Yaskawa INFORM job: SKRZYNIA_5240_0_STOPNI_1OBR.JBI

/JOB
//NAME SKRZYNIA_5240_0_STOPNI_1OBR
///FOLDERNAME 02-SKRZYNIE_JOBS
//POS
///NPOS 629,629,0,49,4,0
///TOOL 0
///POSTYPE PULSE
///PULSE
C00000=1055,-24125,84372,288,19725,204
C00001=1055,-24125,84372,288,19725,204
C00002=0,-15438,65714,0,-68532,0
C00003=25524,-25821,36823,19654,-58495,38520
C00004=25525,-25816,36822,19654,-58489,38517
C00005=24740,-25233,37027,19126,-58082,38651
C00006=23674,-24366,37359,18410,-57511,38837
C00007=23935,-24587,37271,18586,-57653,38791
C00008=22514,-24691,37230,17505,-57481,39152
C00009=26142,-25637,36881,20127,-58504,38350
C00010=24740,-25232,37025,19127,-58082,38646
C00011=24741,-25229,37025,19127,-58082,38646
C00012=24435,-24991,37114,18923,-57922,38699
C00013=23923,-24572,37275,18578,-57647,38788
C00014=24083,-24706,37224,18686,-57733,38759
C00015=22429,-24825,37180,17430,-57534,39178
C00016=25895,-26212,36688,19885,-58747,38460
C00017=25524,-25821,36823,19654,-58495,38520
C00018=23988,-24960,37134,18595,-57837,38812
C00019=22822,-23954,37534,17811,-57199,39017
C00020=22935,-24057,37491,17887,-57262,38997
C00021=20006,-24258,37408,15644,-56932,39751
C00022=24402,-25289,37013,18874,-58060,38740
C00023=22585,-24665,40358,17164,-59622,30036
C00024=23477,-23257,40205,18030,-58646,29630
C00025=22519,-22398,40568,17384,-58125,29795
C00026=22700,-22567,40495,17506,-58225,29764
C00027=19339,-22794,40398,14955,-57865,30607
C00028=24825,-24328,39798,18931,-59350,29401
C00029=32755,-32613,25711,29640,-48730,33694
C00030=25632,-30899,26166,23992,-46203,35378
C00031=24264,-29862,26497,22996,-45413,35639
C00032=24403,-29974,26459,23097,-45496,35612
C00033=20575,-30233,26374,19602,-44891,36810
C00034=26556,-31526,25988,24663,-46720,35206
C00035=30846,-32795,25752,28021,-48338,30427
C00036=24953,-30697,26306,23444,-45946,31743
C00037=23937,-29910,26558,22702,-45353,31936
C00038=24039,-29993,26530,22778,-45414,31916
C00039=20322,-30240,26449,19379,-44834,33080
C00040=25997,-31433,26093,24205,-46535,31545
C00041=26028,-43665,26580,-39946,8682,24640
C00042=27956,-30595,53065,-101898,6609,54413
C00043=26028,-43663,26580,-39944,8677,24639
C00044=38784,-34544,25404,33956,-51320,34445
C00045=29266,-32676,25756,26732,-47889,36488
C00046=25734,-31262,26119,24020,-46377,37252
C00047=24289,-30200,26441,22967,-45549,37525
C00048=24367,-30262,26420,23025,-45594,37511
C00049=20043,-30544,26331,19080,-44922,38860
C00050=26573,-31816,25967,24631,-46839,37095
C00051=27817,-32566,25782,25532,-47502,36865
C00052=26734,-31919,25941,24747,-46925,37065
C00053=24344,-30243,26427,23007,-45578,37515
C00054=24432,-30312,26405,23072,-45630,37498
C00055=20021,-30599,26315,19050,-44944,38872
C00056=26262,-31616,26021,24405,-46667,37153
C00057=27439,-32346,25835,25259,-47302,36935
C00058=27195,-32201,25870,25083,-47172,36980
C00059=24581,-30384,26384,23190,-45695,37464
C00060=24689,-30466,26358,23269,-45758,37444
C00061=20001,-30771,26264,18999,-45026,38899
C00062=26308,-31607,26026,24448,-46671,37139
C00063=28815,-33076,25672,26259,-47996,36678
C00064=25576,-41037,6257,30736,-35041,33971
C00065=22958,-37632,10123,27061,-35370,35326
C00066=22703,-41294,1722,31272,-29953,33282
C00067=19440,-41515,1663,27208,-29122,34832
C00068=25465,-43501,1200,33269,-31905,32752
C00069=87177,-39066,-1236,81808,-72661,19198
C00070=4794,-34097,38974,4189,-31824,-1302
C00071=4794,-34097,38974,4189,13412,-1302
C00072=11237,-37131,38982,-12694,5333,8253
C00073=6591,-33902,35532,5956,-1761,-1932
C00074=10065,-33530,28876,9373,-31104,-3154
C00075=31877,-32319,25770,29025,-48287,33360
C00076=25762,-31514,25979,24006,-46465,34920
C00077=23652,-29939,26460,22464,-45250,35320
C00078=23742,-30013,26436,22530,-45305,35302
C00079=19630,-30281,26348,18756,-44677,36597
C00080=26056,-31710,25928,24219,-46631,34863
C00081=38095,-40136,7813,41252,-44156,24924
C00082=33231,-38681,8176,37792,-41757,25918
C00083=31538,-37640,8473,36716,-40716,26179
C00084=31687,-37737,8444,36811,-40809,26155
C00085=27389,-38154,8322,32773,-39589,27627
C00086=33834,-39023,8084,38175,-42120,25821
C00087=27585,-47842,-289,32095,-40789,28095
C00088=4801,-35772,25187,4593,-28023,-82032
C00089=17634,-23800,39238,9573,-31425,-73339
C00090=17634,-23800,39238,9573,-31425,-73339
C00091=16549,-22464,39800,8390,-30730,-72975
C00092=16684,-22641,39722,8536,-30818,-73021
C00093=16684,-19968,45512,8078,-32771,-72767
C00094=17634,-23800,39238,9573,-31425,-73339
C00095=17837,-21535,44509,9322,-33342,-73155
C00096=17837,-21535,44509,9322,-33342,-73155
C00097=16866,-20378,45014,8305,-32755,-72853
C00098=17032,-20588,44918,8481,-32857,-72905
C00099=17032,-17542,51480,8009,-35060,-72636
C00100=17837,-21535,44509,9322,-33342,-73155
C00101=-20829,-18800,50532,-12466,-37179,-77446
C00102=-19934,-17904,50946,-11618,-36715,-77676
C00103=-20044,-18019,50891,-11723,-36773,-77647
C00104=-20044,-15288,56753,-11218,-38713,-77950
C00105=-20966,-18928,50473,-12596,-37250,-77413
C00106=-20884,-26676,33664,-14451,-31668,-76336
C00107=-20884,-26676,33664,-14451,-31668,-76336
C00108=-19557,-25338,34176,-13080,-30873,-76751
C00109=-19691,-25483,34117,-13220,-30955,-76709
C00110=-19691,-22773,39998,-12506,-32911,-77106
C00111=-20642,-26447,33747,-14206,-31526,-76411
C00112=-33629,-40566,17444,-29603,-33447,-71192
C00113=-33629,-40566,17444,42578,-32312,-84654
C00114=-42160,-31266,16400,42578,-32312,-84654
C00115=-87798,-804,48829,-20188,-26072,-60966
C00116=-76454,-11934,10236,-25964,7954,-64922
C00117=-76448,-11928,10235,-25961,7944,-64914
C00118=-68643,-7759,-23318,-14097,50582,-74897
C00119=-70868,-8793,-8075,-29663,30364,-70765
C00120=-67243,-1968,12282,-49553,26687,-63567
C00121=-68655,-309,14069,-48513,25966,-64203
C00122=-67497,-1678,12591,-49367,26558,-63682
C00123=-71436,-723,2905,-26484,35140,-73726
C00124=-71436,176,6426,-27636,33595,-73066
C00125=-71434,778,8668,-28412,32633,-72624
C00126=-68624,-2689,-85,-28291,36551,-72622
C00127=-99375,3692,5712,40719,48607,-84097
C00128=-94964,4957,10918,40408,44640,-83792
C00129=-93063,6047,12199,39572,43744,-83178
C00130=-94964,4957,10918,40408,44640,-83792
C00131=-94964,5754,13918,41385,43553,-84439
C00132=-94964,4957,10918,40408,44640,-83792
C00133=-90271,-412,-5146,23417,46876,-76529
C00134=-83133,-4088,-8267,6704,41492,-71542
C00135=-83133,-4088,-8267,6704,41492,-71542
C00136=-83133,-4088,-8267,6704,41492,-11598
C00137=-83133,-16026,-8267,6704,41492,-11598
C00138=-83133,-16026,-8267,6704,41492,-11598
C00139=-48225,-19387,30619,3889,32460,-6728
C00140=56943,-39861,25115,1795,-37402,-69601
C00141=29960,-38386,-19607,-115769,-41858,-24264
C00142=65721,-6478,18155,-133323,-22195,3361
C00143=70544,4411,32968,-134868,-18623,4660
C00144=71874,8263,38598,-134556,-17327,4659
C00145=72629,9390,40002,-135279,-16924,5107
C00146=71441,7638,37831,-134139,-17555,4406
C00147=77146,8888,25050,-166574,-32612,18372
C00148=77146,10029,28643,-166204,-31014,18167
C00149=77146,11198,32202,-165803,-29459,17947
C00150=75508,4678,16951,-165715,-35157,17778
C00151=68680,12216,24468,-164340,-40455,-13359
C00152=68362,12845,25743,-164045,-40097,-13561
C00153=68362,13700,28585,-163752,-38808,-13742
C00154=68362,12845,25743,-164045,-40097,-13561
C00155=64993,-1168,28876,-102971,-10760,-49875
C00156=63888,481,30670,-102324,-11438,-50313
C00157=64993,-1168,28876,-102971,-10760,-49875
C00158=4264,-34194,25387,4006,-26954,-29436
C00159=4264,-34194,25387,4006,-26954,-81856
C00160=17634,-23800,39238,9573,-31425,-73339
C00161=17837,-27228,32238,10495,-29236,-73805
C00162=17837,-21535,44509,9322,-33342,-73155
C00163=17548,-20734,45666,8935,-33511,-73021
C00164=-20829,-18800,50532,-12466,-37179,-77446
C00165=-20884,-20901,46110,-12960,-35762,-77182
C00166=-20884,-26676,33664,-14451,-31668,-76336
C00167=-20624,-26699,33167,-14265,-31320,-76369
C00168=-33629,-40566,17444,-29603,-33447,-71192
C00169=-33629,-40566,17444,42578,-32312,-84654
C00170=-42160,-31266,16400,42578,-32312,-84654
C00171=-87798,-804,48829,-20188,-26072,-60966
C00172=-76454,-11934,10236,-25964,7954,-64922
C00173=-76448,-11928,10235,-25961,7944,-64914
C00174=-68643,-7759,-23318,-14097,50582,-74897
C00175=-70868,-8793,-8075,-29663,30364,-70765
C00176=-67243,-1968,12282,-49553,26687,-63567
C00177=-68655,-309,14069,-48513,25966,-64203
C00178=-67497,-1678,12591,-49367,26558,-63682
C00179=-71436,-723,2905,-26484,35140,-73726
C00180=-71436,176,6426,-27636,33595,-73066
C00181=-71434,778,8668,-28412,32633,-72624
C00182=-68624,-2689,-85,-28291,36551,-72622
C00183=-99375,3692,5712,40719,48607,-84097
C00184=-94964,4957,10918,40408,44640,-83792
C00185=-93063,6047,12199,39572,43744,-83178
C00186=-94964,4957,10918,40408,44640,-83792
C00187=-94964,5754,13918,41385,43553,-84439
C00188=-94964,4957,10918,40408,44640,-83792
C00189=-90271,-412,-5146,23417,46876,-76529
C00190=-83133,-4088,-8267,6704,41492,-71542
C00191=-83133,-4088,-8267,6704,41492,-71542
C00192=-83133,-4088,-8267,6704,41492,-11598
C00193=-83133,-16026,-8267,6704,41492,-11598
C00194=-83133,-16026,-8267,6704,41492,-11598
C00195=-48225,-19387,30619,3889,32460,-6728
C00196=56943,-39861,25115,1795,-37402,-69601
C00197=29960,-38386,-19607,-115769,-41858,-24264
C00198=65721,-6478,18155,-133323,-22195,3361
C00199=70544,4411,32968,-134868,-18623,4660
C00200=71874,8263,38598,-134556,-17327,4659
C00201=72629,9390,40002,-135279,-16924,5107
C00202=71441,7638,37831,-134139,-17555,4406
C00203=77146,8888,25050,-166574,-32612,18372
C00204=77146,10029,28643,-166204,-31014,18167
C00205=77146,11198,32202,-165803,-29459,17947
C00206=75508,4678,16951,-165715,-35157,17778
C00207=68680,12216,24468,-164340,-40455,-13359
C00208=68362,12845,25743,-164045,-40097,-13561
C00209=68362,13700,28585,-163752,-38808,-13742
C00210=68362,12845,25743,-164045,-40097,-13561
C00211=64993,-1168,28876,-102971,-10760,-49875
C00212=63888,481,30670,-102324,-11438,-50313
C00213=64993,-1168,28876,-102971,-10760,-49875
C00214=58588,-14653,4620,-120782,-19611,-35794
C00215=29960,-38386,-19607,-115769,-41858,-24264
C00216=56943,-39861,25115,1795,-37402,-69601
C00217=-1002,-39861,25115,1795,-37402,-69601
C00218=-1001,-39858,25114,1795,-37402,0
C00219=6591,-33902,35532,5956,-1761,-1932
C00220=6592,-33900,35531,103508,-35512,-26314
C00221=-99253,-13690,44082,59847,13407,-31313
C00222=-85045,-36869,-4353,28502,-22832,-52282
C00223=-92346,-18713,13565,21110,-22545,-55257
C00224=-85370,-14218,16934,32905,-23649,-60330
C00225=-84150,-13282,17685,34842,-23935,-61163
C00226=-82877,-12536,18624,36445,-24482,-61818
C00227=-84150,-13282,17685,34842,-23935,-61163
C00228=-85467,-11480,19558,33086,-23405,-60436
C00229=-84150,-13282,17685,34842,-23935,-61163
C00230=-85732,-21202,11427,30682,-24763,-59235
C00231=-84559,-15616,15722,33768,-24118,-60665
C00232=-84150,-13282,17685,34842,-23935,-61163
C00233=-83260,-12880,18034,36130,-24218,-61709
C00234=-84150,-13282,17685,34842,-23935,-61163
C00235=-85365,-11775,19006,33430,-23307,-60600
C00236=-84150,-13282,17685,34842,-23935,-61163
C00237=-85786,-16909,14677,31743,-23900,-59790
C00238=-84150,-13282,17685,34842,-23935,-61163
C00239=-83215,-12861,18051,36194,-24233,-61735
C00240=-84150,-13282,17685,34842,-23935,-61163
C00241=-85327,-11825,18959,33476,-23327,-60618
C00242=-84150,-13282,17685,34842,-23935,-61163
C00243=-87841,-18519,13420,28367,-23534,-58339
C00244=-84150,-13282,17685,34842,-23935,-61163
C00245=-83292,-12894,18020,36083,-24208,-61688
C00246=-84150,-13282,17685,34842,-23935,-61163
C00247=-85185,-12008,18799,33646,-23400,-60687
C00248=-84150,-13282,17685,34842,-23935,-61163
C00249=-86371,-18277,13606,30568,-23951,-59265
C00250=-84345,-13370,17612,34554,-23873,-61041
C00251=-83240,-12871,18042,36158,-24225,-61720
C00252=-84345,-13370,17612,34554,-23873,-61041
C00253=-85365,-12110,18711,33368,-23345,-60568
C00254=-84345,-13370,17612,34554,-23873,-61041
C00255=-86191,-19647,12567,30467,-24278,-59187
C00256=-84345,-13372,17610,34552,-23873,-61039
C00257=-83096,-12807,18098,36363,-24268,-61804
C00258=-84345,-13372,17610,34552,-23873,-61039
C00259=-85268,-12232,18600,33480,-23393,-60612
C00260=-84345,-13372,17610,34552,-23873,-61039
C00261=-84814,-16043,15376,33312,-24093,-60464
C00262=-84104,-13265,17702,34906,-23948,-61189
C00263=-82960,-12743,18153,36555,-24313,-61887
C00264=-84104,-13265,17702,34906,-23948,-61189
C00265=-84979,-12194,18635,33901,-23496,-60788
C00266=-84104,-13265,17702,34906,-23948,-61189
C00267=-86610,-16845,14732,30573,-23614,-59301
C00268=-84104,-13265,17702,34906,-23948,-61189
C00269=-82793,-12667,18222,36790,-24370,-61986
C00270=-84104,-13265,17702,34906,-23948,-61189
C00271=-84888,-12305,18537,34004,-23540,-60830
C00272=-84104,-13265,17702,34906,-23948,-61189
C00273=-83806,-19585,12613,33764,-25080,-60559
C00274=-83675,-13072,17868,35530,-24083,-61453
C00275=-82553,-12556,18319,37130,-24451,-62127
C00276=-83675,-13072,17868,35530,-24083,-61453
C00277=-84378,-12223,18610,34735,-23716,-61138
C00278=-83675,-13072,17868,35530,-24083,-61453
C00279=-87149,-17993,13826,29513,-23647,-58830
C00280=-84104,-13265,17702,34906,-23948,-61189
C00281=-82640,-12594,18285,37014,-24425,-62079
C00282=-84104,-13265,17702,34906,-23948,-61189
C00283=-84792,-12429,18430,34119,-23592,-60877
C00284=-84104,-13265,17702,34906,-23948,-61189
C00285=-83583,-9185,30892,23668,-36042,-57025
C00286=-85789,-8328,35795,20592,-37093,-55378
C00287=-85786,-16735,14816,31782,-23869,-59812
C00288=-84103,-13263,17702,34906,-23947,-61191
C00289=-83225,-12865,18046,36177,-24227,-61729
C00290=-84103,-13263,17702,34906,-23947,-61191
C00291=-84774,-12447,18412,34138,-23599,-60886
C00292=-84103,-13263,17702,34906,-23947,-61191
C00293=-86149,-16246,6730,18897,-35239,-57128
C00294=-86244,-15289,7532,18875,-35060,-57127
C00295=-85361,-14893,7870,19824,-35193,-57574
C00296=-86244,-15289,7532,18875,-35060,-57127
C00297=-86889,-14409,8282,18264,-34784,-56850
C00298=-86244,-15289,7532,18875,-35060,-57127
C00299=-90262,-21765,2389,14114,-35574,-54847
C00300=-90262,-21765,2389,28730,-17672,-54847
C00301=-89967,-19086,25635,28730,-17672,-54847
C00302=568,-24029,84339,168,19981,112
C00303=568,-24677,83015,164,20405,113
C00304=101153,-24598,83176,165,20353,113
C00305=101153,-24598,83176,165,20353,113
C00306=89967,-19086,25635,-28730,-17672,54847
C00307=90262,-21765,2389,-28730,-17672,54847
C00308=86932,-18662,4771,-17876,-35519,56628
C00309=86578,-15436,7408,-18515,-35011,56957
C00310=85428,-14922,7844,-19753,-35183,57541
C00311=84405,-14447,8250,-20842,-35348,58054
C00312=85428,-14922,7844,-19753,-35183,57541
C00313=86134,-13973,8661,-19091,-34881,57237
C00314=85428,-14922,7844,-19753,-35183,57541
C00315=85786,-16735,14816,-31782,-23869,59812
C00316=83514,-12996,17929,-35760,-24132,61552
C00317=82296,-12429,18424,-37488,-24534,62281
C00318=83514,-12996,17929,-35760,-24132,61552
C00319=84266,-12085,18725,-34910,-23738,61214
C00320=83514,-12996,17929,-35760,-24132,61552
C00321=87323,-6914,39851,-18853,-38149,44508
C00322=83118,-12818,18089,-36330,-24263,61791
C00323=81969,-12276,18566,-37944,-24648,62472
C00324=83118,-12818,18089,-36330,-24263,61791
C00325=83927,-11846,18941,-35423,-23842,61433
C00326=83118,-12818,18089,-36330,-24263,61791
C00327=83806,-19585,12613,-33764,-25080,60559
C00328=83148,-12832,18077,-36287,-24254,61773
C00329=81889,-12236,18598,-38058,-24676,62520
C00330=83148,-12832,18077,-36287,-24254,61773
C00331=83900,-11930,18867,-35446,-23862,61440
C00332=83148,-12832,18077,-36287,-24254,61773
C00333=86610,-16845,14732,-30573,-23614,59301
C00334=82493,-13239,17725,-37070,-24559,62089
C00335=81442,-12739,18159,-38529,-24915,62703
C00336=82493,-13239,17725,-37070,-24559,62089
C00337=83435,-12133,18689,-36040,-24063,61682
C00338=82493,-13239,17725,-37070,-24559,62089
C00339=84814,-16043,15376,-33312,-24093,60464
C00340=82555,-13613,17404,-36910,-24580,62015
C00341=81369,-13053,17885,-38558,-24979,62709
C00342=82555,-13613,17404,-36910,-24580,62015
C00343=83568,-12431,18429,-35805,-24046,61580
C00344=82555,-13613,17404,-36910,-24580,62015
C00345=86191,-19647,12567,-30467,-24278,59187
C00346=82500,-13648,17375,-36975,-24607,62039
C00347=81594,-13224,17740,-38236,-24911,62571
C00348=82500,-13648,17375,-36975,-24607,62039
C00349=83449,-12543,18332,-35941,-24104,61633
C00350=82500,-13648,17375,-36975,-24607,62039
C00351=86371,-18277,13606,-30568,-23951,59265
C00352=82904,-13790,17251,-36416,-24470,61808
C00353=81796,-13275,17692,-37971,-24838,62464
C00354=82904,-13790,17251,-36416,-24470,61808
C00355=83696,-12867,18046,-35547,-24051,61466
C00356=82904,-13790,17251,-36416,-24470,61808
C00357=87841,-18519,13420,-28367,-23534,58339
C00358=82748,-13879,17174,-36603,-24542,61883
C00359=81789,-13434,17554,-37946,-24861,62449
C00360=82748,-13879,17174,-36603,-24542,61883
C00361=83603,-12888,18026,-35668,-24086,61514
C00362=82748,-13879,17174,-36603,-24542,61883
C00363=85786,-16909,14677,-31743,-23900,59790
C00364=82339,-14116,16972,-37087,-24733,62079
C00365=81557,-13752,17280,-38171,-24994,62536
C00366=82339,-14116,16972,-37087,-24733,62079
C00367=83390,-12909,18006,-35951,-24172,61633
C00368=82339,-14116,16972,-37087,-24733,62079
C00369=85732,-21202,11427,-30682,-24763,59235
C00370=82398,-14365,16763,-36952,-24745,62014
C00371=81340,-13876,17176,-38416,-25096,62632
C00372=82398,-14365,16763,-36952,-24745,62014
C00373=83629,-12951,17972,-35620,-24090,61491
C00374=82398,-14365,16763,-36952,-24745,62014
C00375=92346,-18713,13565,-21110,-22545,55257
C00376=82794,-13980,17083,-36511,-24538,61844
C00377=81697,-13472,17516,-38043,-24902,62488
C00378=82794,-13980,17083,-36511,-24538,61844
C00379=83767,-12847,18056,-35444,-24023,61424
C00380=82794,-13980,17083,-36511,-24538,61844
C00381=85045,-36869,-4353,-28502,-22832,52282
C00382=69856,-53931,-13446,-33557,-28911,29591
C00383=73943,-28815,39553,-16801,-45089,19004
C00384=0,-24029,84339,0,19981,0
C00385=0,-24029,84339,0,19981,0
C00386=0,-52280,40443,0,6876,0
C00387=63961,-36661,14391,66570,-58199,13439
C00388=51209,-38551,620,65071,-48478,10741
C00389=46952,-37885,872,62997,-46041,11191
C00390=46598,-37935,846,62778,-45862,11259
C00391=54160,-39955,137,66075,-50361,10746
C00392=0,-52280,40443,0,6876,0
C00393=0,-52280,40443,0,6876,0
C00394=42978,-45587,7631,48214,-41849,18034
C00395=36694,-44945,-1657,49443,-34807,15750
C00396=45238,-39007,-3596,70255,-41437,11463
C00397=45059,-39151,-3508,69830,-41334,11649
C00398=32474,-45233,-13338,65386,-28486,22104
C00399=59828,-44646,-5405,72855,-48572,12139
C00400=0,-38761,66314,0,-763,0
C00401=0,-44757,54667,0,2744,0
C00402=40382,-38226,12225,48505,-40693,16039
C00403=55481,-27484,23768,62968,-54833,11978
C00404=49623,-26525,24220,59800,-51818,12584
C00405=49591,-31309,12277,55066,-55958,13102
C00406=55330,-33748,11238,57660,-59334,12681
C00407=78664,-24436,10378,82837,-79111,12029
C00408=75189,-23065,11287,81851,-76948,11927
C00409=75189,-45249,11287,81851,-38847,11927
C00410=29880,-45249,11287,43145,-11324,11927
C00411=0,-24029,84339,0,19981,0
C00412=0,-24026,84338,1,19977,2
C00413=4264,-34194,25387,4006,-26954,-29436
C00414=4264,-34194,25387,4006,-26954,-81856
C00415=-21478,-27798,32214,-15234,-31599,-76056
C00416=-19679,-23059,39354,-12567,-32689,-77067
C00417=16724,-20576,44291,8212,-32395,-72836
C00418=21329,-26386,39716,13285,-34016,-74401
C00419=-23778,-26243,38799,-16502,-35132,-75964
C00420=-20075,-15782,55752,-11329,-38404,-77896
C00421=16874,-17447,51356,7863,-34895,-72604
C00422=18580,-28601,30698,11472,-29284,-74138
C00423=6126,-41331,18955,6697,-26557,-30383
C00424=1,-24024,84337,2,19973,1
C00425=-64243,-26178,31107,-39513,40312,-5844
C00426=-72148,3973,56008,-35470,42045,-10522
C00427=-72090,16396,76301,-42067,35650,-6519
C00428=-69388,15725,61378,-31740,35177,-8719
C00429=-69127,27099,75569,-32744,34250,-8088
C00430=-67573,2495,11285,-21767,57629,-15193
C00431=-77819,19629,29798,-10454,63174,-20704
C00432=-72990,23583,14304,-10735,77209,-20379
C00433=-74593,38003,46707,-11043,65751,-19814
C00434=-73236,38943,48295,-11400,65557,-19316
C00435=-73329,42107,51779,-6346,67443,-19636
C00436=-87142,34654,46174,17622,63862,-25393
C00437=-87240,36727,48611,18897,66604,-25032
C00438=-99033,21517,12213,24947,79702,-26203
C00439=-91500,-14196,-34781,24472,81625,-22832
C00440=-100472,-45007,-27818,8167,67201,-29302
C00441=0,-36642,16905,0,48372,0
C00442=66009,-61997,-62105,21406,63483,18379
C00443=97242,-23579,-39442,10179,68876,30321
C00444=73684,-7073,-17511,24638,68131,29022
C00445=59136,7235,6676,33270,66602,27507
C00446=54816,14937,6234,39741,69494,31070
C00447=54365,20668,19279,41017,66202,29418
C00448=64503,4223,2857,29650,48528,26647
C00449=75622,3202,-3149,3890,49494,34281
C00450=88036,13177,2413,-18568,66573,35876
C00451=90462,21593,10123,-22613,76266,34479
C00452=92450,29224,20002,-25750,81642,33727
C00453=94949,8131,-12163,-20291,74229,36861
C00454=94949,8084,-13484,-20215,75047,36712
C00455=70412,-34016,-52305,-11724,65624,29757
C00456=18580,-28601,30698,11472,-29284,-74138
C00457=-23778,-26243,38799,-16502,-35132,-75964
C00458=18580,-28601,30698,11472,-29284,-74138
C00459=4264,-34194,25387,4006,-26954,-81856
C00460=4264,-34194,25387,4006,-26954,-29436
C00461=1,-24024,84337,2,19973,1
C00462=-64243,-26178,31107,-39513,40312,-5844
C00463=-72148,3973,56008,-35470,42045,-10522
C00464=-72090,16396,76301,-42067,35650,-6519
C00465=-69388,15725,61378,-31740,35177,-8719
C00466=-69127,27099,75569,-32744,34250,-8088
C00467=-67573,2495,11285,-21767,57629,-15193
C00468=-77819,19629,29798,-10454,63174,-20704
C00469=-72990,23583,14304,-10735,77209,-20379
C00470=-74593,38003,46707,-11043,65751,-19814
C00471=-73236,38943,48295,-11400,65557,-19316
C00472=-73329,42107,51779,-6346,67443,-19636
C00473=-87142,34654,46174,17622,63862,-25393
C00474=-87240,36727,48611,18897,66604,-25032
C00475=-99033,21517,12213,24947,79702,-26203
C00476=-91500,-14196,-34781,24472,81625,-22832
C00477=-100472,-45007,-27818,8167,67201,-29302
C00478=0,-36642,16905,0,48372,0
C00479=66009,-61997,-62105,21406,63483,18379
C00480=97242,-23579,-39442,10179,68876,30321
C00481=73684,-7073,-17511,24638,68131,29022
C00482=59136,7235,6676,33270,66602,27507
C00483=54816,14937,6234,39741,69494,31070
C00484=54365,20668,19279,41017,66202,29418
C00485=64503,4223,2857,29650,48528,26647
C00486=75622,3202,-3149,3890,49494,34281
C00487=88036,13177,2413,-18568,66573,35876
C00488=90462,21593,10123,-22613,76266,34479
C00489=92450,29224,20002,-25750,81642,33727
C00490=94949,8131,-12163,-20291,74229,36861
C00491=94949,8084,-13484,-20215,75047,36712
C00492=70412,-34016,-52305,-11724,65624,29757
C00493=44268,-30306,-1568,-7370,48673,18708
C00494=1,-24024,84337,2,19973,1
C00495=1,-24024,84337,2,19973,1
C00496=3796,-57671,22373,2336,-25309,-753
C00497=52632,-34554,16626,51161,-63050,5622
C00498=59461,-32779,9832,66317,-58406,17312
C00499=52745,-27759,19165,60340,-56543,14824
C00500=51596,-17381,41670,51728,-64721,19335
C00501=62932,-33588,12189,66848,-61063,18031
C00502=55481,-27484,23768,62968,-54833,11978
C00503=57132,-27695,23671,63846,-55681,11818
C00504=51865,-26731,24121,61082,-52936,12300
C00505=51802,-31418,12227,56278,-57054,12744
C00506=55330,-33748,11238,57660,-59334,12681
C00507=1,-24024,84337,2,19973,1
C00508=1,-24024,84337,2,19973,1
C00509=57188,-41777,19973,48132,-58706,4905
C00510=55566,-48748,-16991,79805,-45048,-6941
C00511=49908,-48716,-25784,90749,-41340,-3650
C00512=44141,-47261,-25474,90786,-37676,-4452
C00513=43373,-46910,-25348,90885,-37191,-4606
C00514=55479,-50244,-26473,91085,-44870,-3042
C00515=12119,-24859,71505,13236,4440,2633
C00516=-91085,-34291,10385,1908,-24348,-42097
C00517=-86191,-19647,12567,30467,-24278,-59187
C00518=-99148,-11667,19101,-13975,-20192,-40187
C00519=-98206,-11518,19604,-10142,-20308,-41629
C00520=-99474,-20389,12397,-11593,-22150,-41069
C00521=0,-52280,40443,0,6876,0
C00522=85348,-24204,23536,-13963,-15515,44275
C00523=84670,-17015,14597,-33277,-24304,60423
C00524=96971,-12584,18294,8365,-19955,42614
C00525=97182,-12918,18001,8747,-20027,42449
C00526=96230,-24528,9149,6144,-22576,43630
C00527=0,-52280,40443,0,6876,0
C00528=0,-52280,40443,0,6876,0
C00529=-90140,-60305,18108,-2708,1721,-7625
C00530=-95594,-27428,6866,-4663,-19832,-42154
C00531=-99356,-13410,18355,-15385,-17730,-37479
C00532=-99405,-10878,20508,-15853,-17333,-37255
C00533=-99132,-10804,20575,-15274,-17279,-37502
C00534=-99132,-3482,39129,-10940,-24351,-39674
C00535=-98851,-3328,38974,-10588,-24101,-39807
C00536=-100183,-18601,14070,-16273,-18800,-37146
C00537=-90140,-60305,18108,-2708,1721,-7625
C00538=0,-52280,40443,0,6876,0
C00539=84259,-57935,27522,-3761,3673,6310
C00540=86507,-39672,4297,-27618,-16640,46340
C00541=70477,-27878,7073,-45786,-32339,64941
C00542=84043,-16293,15174,-34312,-24409,60872
C00543=100395,-12639,18246,19464,-20904,37830
C00544=99154,-17369,4403,32227,-9753,28926
C00545=99154,-17369,4403,32227,-9753,28926
C00546=98946,-17182,4556,31649,-9649,29182
C00547=100388,-17987,13832,15751,-21517,39479
C00548=86507,-39672,4297,-27618,-16640,46340
C00549=84259,-57935,27522,-3761,3673,6310
C00550=0,-52280,40443,0,6876,0
C00551=0,-27933,77061,0,20812,0
C00552=0,-27933,77061,0,20812,0
C00553=0,-52280,40443,0,6876,0
C00554=-91970,-60791,14435,-3343,512,-9412
C00555=-99196,-15868,16098,-13748,-19297,-38710
C00556=-99196,-15868,16098,-13748,-19297,-38710
C00557=-99196,-15868,16098,-13748,-19297,-38710
C00558=-85815,-11758,19597,31748,-21097,-58265
C00559=-87383,-11883,19487,26986,-20206,-56250
C00560=-99562,-16264,15781,-14410,-19427,-38431
C00561=-99196,-15868,16098,-13748,-19297,-38710
C00562=-91970,-60791,14435,-3343,512,-9412
C00563=0,-52280,40443,0,6876,0
C00564=91083,-60784,14823,-9043,-825,15173
C00565=83869,-19403,12921,-33769,-24740,60260
C00566=83869,-19403,12921,-33769,-24740,60260
C00567=83420,-14897,16486,-35538,-24144,61113
C00568=90535,-11845,19652,-14037,-20800,51549
C00569=90317,-11662,19878,-14346,-20882,51648
C00570=95871,-14889,15992,4901,-19605,43825
C00571=83869,-19403,12921,-33769,-24740,60260
C00572=91083,-60784,14823,-9043,-825,15173
C00573=0,-52280,40443,0,6876,0
C00574=-91526,-60598,16699,7584,176,-13289
C00575=-94392,-6553,48683,5805,-47321,-49764
C00576=-88951,-345,54953,10686,-47392,-51569
C00577=-88172,5833,62122,11322,-47753,-51785
C00578=-90949,-14015,9500,8834,-34399,-51934
C00579=-84917,-15593,15742,33275,-23984,-60461
C00580=-81669,-15982,15425,37506,-25258,-62202
C00581=-79867,-25377,9541,37586,-25936,-59971
C00582=-91415,-60262,16631,7870,-73,-13734
C00583=24,-24029,84339,7,19981,5
C00584=160,-24029,84339,47,19981,32
C00585=99096,-24029,84339,47,19981,32
C00586=99096,-24029,84339,47,19981,32
C00587=89967,-19086,25635,-28730,-17672,54847
C00588=85786,-16735,14816,-31782,-23869,59812
C00589=83492,-14473,16674,-35480,-24338,61406
C00590=82709,-11470,19305,-37370,-24374,62232
C00591=85293,-13629,8874,-19696,-34851,57583
C00592=85505,-16299,6686,-19564,-35388,57437
C00593=89967,-19086,25635,-28730,-17672,54847
C00594=568,-24029,84339,168,19981,112
C00595=568,-24029,84339,168,19981,112
C00596=-91970,-60791,14435,-3343,512,-9412
C00597=-86948,-23217,10819,28314,-23349,-56438
C00598=-85895,-16522,15767,31843,-22281,-58087
C00599=-93643,1708,52973,2937,-38210,-34777
C00600=-93409,-737,47229,3345,-36106,-34967
C00601=-86145,-24679,9854,29028,-23971,-56682
C00602=-100471,-58311,4157,14142,-4822,-27614
C00603=-68517,-58311,4157,14142,-4822,-27614
C00604=0,-52280,40443,0,6876,0
C00605=91083,-60784,14823,-9043,-825,15173
C00606=83869,-19403,12921,-33769,-24740,60260
C00607=82620,-18743,14708,-32942,-26226,58979
C00608=83315,-11405,20766,-33572,-24860,59408
C00609=83326,-11144,20997,-33599,-24827,59423
C00610=84798,-22668,11879,-29033,-26372,57255
C00611=91083,-60784,14823,-9043,-825,15173
C00612=0,-52280,40443,0,6876,0
C00613=-6369,-39206,65423,-4801,-482,2563
C00614=-97287,-29142,12714,-8673,-22288,-37832
C00615=-86191,-19647,12567,30467,-24278,-59187
C00616=-85671,-16302,15857,30808,-24404,-58999
C00617=-99965,-10410,22406,-14600,-22538,-38834
C00618=-95758,-10871,21797,-1120,-21702,-44724
C00619=-87910,-17792,15835,25414,-24996,-56048
C00620=-97287,-29142,12714,-8673,-22288,-37832
C00621=0,-52280,40443,0,6876,0
C00622=92301,-25634,22749,2368,-15645,37646
C00623=83738,-18329,13570,-34202,-24868,60772
C00624=90096,-13099,18146,-15422,-20883,52700
C00625=93330,-13245,17928,-4627,-20146,48105
C00626=80226,-20465,12178,-39626,-27411,62762
C00627=92301,-25634,22749,2368,-15645,37646
C00628=0,-52280,40443,0,6876,0
BC00000=413138
BC00001=413138
BC00002=413138
BC00003=413134
BC00004=283607
BC00005=283607
BC00006=283607
BC00007=283607
BC00008=283607
BC00009=283607
BC00010=283606
BC00011=344572
BC00012=344572
BC00013=344572
BC00014=344572
BC00015=344572
BC00016=344572
BC00017=413134
BC00018=413134
BC00019=413134
BC00020=413134
BC00021=413134
BC00022=413134
BC00023=474623
BC00024=474628
BC00025=474628
BC00026=474628
BC00027=474628
BC00028=474628
BC00029=522849
BC00030=522849
BC00031=522849
BC00032=522849
BC00033=522849
BC00034=522849
BC00035=586045
BC00036=586045
BC00037=586045
BC00038=586045
BC00039=586045
BC00040=586045
BC00041=479622
BC00042=618860
BC00043=673957
BC00044=655410
BC00045=655410
BC00046=655410
BC00047=655410
BC00048=655410
BC00049=655410
BC00050=655410
BC00051=708270
BC00052=708270
BC00053=708270
BC00054=708270
BC00055=708270
BC00056=708270
BC00057=770184
BC00058=770184
BC00059=770184
BC00060=770184
BC00061=770184
BC00062=770184
BC00063=823730
BC00064=829967
BC00065=829969
BC00066=829970
BC00067=829970
BC00068=829970
BC00069=838761
BC00070=740349
BC00071=687700
BC00072=771943
BC00073=861898
BC00074=881669
BC00075=901229
BC00076=901229
BC00077=901229
BC00078=901229
BC00079=901229
BC00080=901229
BC00081=949836
BC00082=949836
BC00083=949836
BC00084=949836
BC00085=949836
BC00086=949836
BC00087=980558
BC00088=926513
BC00089=941874
BC00090=941874
BC00091=941874
BC00092=941874
BC00093=941874
BC00094=941874
BC00095=946320
BC00096=946320
BC00097=946320
BC00098=946320
BC00099=946320
BC00100=946320
BC00101=946320
BC00102=946320
BC00103=946320
BC00104=946320
BC00105=946320
BC00106=946320
BC00107=946320
BC00108=946320
BC00109=946320
BC00110=946320
BC00111=946320
BC00112=946320
BC00113=946320
BC00114=946320
BC00115=946320
BC00116=946320
BC00117=964072
BC00118=975158
BC00119=991862
BC00120=991862
BC00121=991862
BC00122=991862
BC00123=991862
BC00124=991862
BC00125=991863
BC00126=991863
BC00127=991863
BC00128=991863
BC00129=991863
BC00130=991863
BC00131=991863
BC00132=991863
BC00133=982240
BC00134=967606
BC00135=942341
BC00136=942341
BC00137=942341
BC00138=909159
BC00139=874726
BC00140=946320
BC00141=946320
BC00142=946320
BC00143=962534
BC00144=967695
BC00145=967695
BC00146=967695
BC00147=967695
BC00148=967695
BC00149=967695
BC00150=967695
BC00151=967695
BC00152=967695
BC00153=967695
BC00154=967695
BC00155=967695
BC00156=967695
BC00157=967695
BC00158=926513
BC00159=957235
BC00160=941874
BC00161=941874
BC00162=946320
BC00163=946320
BC00164=946320
BC00165=946320
BC00166=946320
BC00167=946320
BC00168=946320
BC00169=946320
BC00170=946320
BC00171=946320
BC00172=946320
BC00173=964072
BC00174=975158
BC00175=991862
BC00176=991862
BC00177=991862
BC00178=991862
BC00179=991862
BC00180=991862
BC00181=991863
BC00182=991863
BC00183=991863
BC00184=991863
BC00185=991863
BC00186=991863
BC00187=991863
BC00188=991863
BC00189=982240
BC00190=967606
BC00191=942341
BC00192=942341
BC00193=942341
BC00194=909159
BC00195=874726
BC00196=946320
BC00197=946320
BC00198=946320
BC00199=962534
BC00200=967695
BC00201=967695
BC00202=967695
BC00203=967695
BC00204=967695
BC00205=967695
BC00206=967695
BC00207=967695
BC00208=967695
BC00209=967695
BC00210=967695
BC00211=967695
BC00212=967695
BC00213=967695
BC00214=962182
BC00215=946320
BC00216=915598
BC00217=915598
BC00218=930961
BC00219=861898
BC00220=861901
BC00221=861901
BC00222=931504
BC00223=963634
BC00224=963631
BC00225=963631
BC00226=963631
BC00227=963631
BC00228=963631
BC00229=963631
BC00230=902188
BC00231=902188
BC00232=902188
BC00233=902188
BC00234=902188
BC00235=902188
BC00236=902188
BC00237=840744
BC00238=840744
BC00239=840744
BC00240=840744
BC00241=840744
BC00242=840744
BC00243=779300
BC00244=779300
BC00245=779300
BC00246=779300
BC00247=779300
BC00248=779300
BC00249=717855
BC00250=717855
BC00251=717855
BC00252=717855
BC00253=717855
BC00254=717855
BC00255=656405
BC00256=656405
BC00257=656405
BC00258=656405
BC00259=656405
BC00260=656405
BC00261=594961
BC00262=594961
BC00263=594961
BC00264=594961
BC00265=594961
BC00266=594961
BC00267=533517
BC00268=533517
BC00269=533517
BC00270=533517
BC00271=533517
BC00272=533517
BC00273=472073
BC00274=472073
BC00275=472073
BC00276=472073
BC00277=472073
BC00278=472073
BC00279=410629
BC00280=410629
BC00281=410629
BC00282=410629
BC00283=410629
BC00284=410629
BC00285=410629
BC00286=349186
BC00287=349186
BC00288=349186
BC00289=349186
BC00290=349186
BC00291=349186
BC00292=349186
BC00293=336469
BC00294=336469
BC00295=336469
BC00296=336469
BC00297=336469
BC00298=336469
BC00299=336469
BC00300=336469
BC00301=336469
BC00302=336469
BC00303=511557
BC00304=512005
BC00305=363797
BC00306=336469
BC00307=336469
BC00308=337415
BC00309=337415
BC00310=337415
BC00311=337415
BC00312=337415
BC00313=337415
BC00314=337415
BC00315=349186
BC00316=350137
BC00317=350137
BC00318=350137
BC00319=350137
BC00320=350137
BC00321=410629
BC00322=411580
BC00323=411580
BC00324=411580
BC00325=411580
BC00326=411580
BC00327=472073
BC00328=473025
BC00329=473025
BC00330=473025
BC00331=473025
BC00332=473025
BC00333=533517
BC00334=534468
BC00335=534468
BC00336=534468
BC00337=534468
BC00338=534468
BC00339=594961
BC00340=594961
BC00341=594961
BC00342=594961
BC00343=594961
BC00344=594961
BC00345=656405
BC00346=657350
BC00347=657350
BC00348=657350
BC00349=657350
BC00350=657350
BC00351=717855
BC00352=718799
BC00353=718799
BC00354=718799
BC00355=718799
BC00356=718799
BC00357=779300
BC00358=780245
BC00359=780245
BC00360=780245
BC00361=780245
BC00362=780245
BC00363=840744
BC00364=841691
BC00365=841691
BC00366=841691
BC00367=841691
BC00368=841691
BC00369=902188
BC00370=903136
BC00371=903136
BC00372=903136
BC00373=903136
BC00374=903136
BC00375=963634
BC00376=963633
BC00377=963633
BC00378=963633
BC00379=963633
BC00380=963633
BC00381=931504
BC00382=861901
BC00383=861901
BC00384=769966
BC00385=769966
BC00386=716865
BC00387=660977
BC00388=660977
BC00389=660977
BC00390=717171
BC00391=717171
BC00392=716865
BC00393=796033
BC00394=895097
BC00395=895097
BC00396=895097
BC00397=945882
BC00398=955598
BC00399=945882
BC00400=840120
BC00401=538973
BC00402=485226
BC00403=456696
BC00404=456696
BC00405=417276
BC00406=417276
BC00407=493986
BC00408=514306
BC00409=514306
BC00410=514306
BC00411=493986
BC00412=797003
BC00413=895791
BC00414=895791
BC00415=946320
BC00416=946320
BC00417=941873
BC00418=936107
BC00419=931618
BC00420=946320
BC00421=946320
BC00422=945548
BC00423=949140
BC00424=797001
BC00425=812363
BC00426=812363
BC00427=869073
BC00428=888959
BC00429=913898
BC00430=945830
BC00431=945830
BC00432=973339
BC00433=973339
BC00434=973339
BC00435=973340
BC00436=973340
BC00437=973341
BC00438=973341
BC00439=973341
BC00440=887999
BC00441=846597
BC00442=930137
BC00443=969257
BC00444=969258
BC00445=969258
BC00446=999505
BC00447=999505
BC00448=999505
BC00449=999505
BC00450=999505
BC00451=999508
BC00452=999508
BC00453=999508
BC00454=973102
BC00455=973102
BC00456=895791
BC00457=900237
BC00458=895791
BC00459=895791
BC00460=895791
BC00461=797001
BC00462=812363
BC00463=812363
BC00464=869073
BC00465=888959
BC00466=913898
BC00467=945830
BC00468=945830
BC00469=973339
BC00470=973339
BC00471=973339
BC00472=973340
BC00473=973340
BC00474=973341
BC00475=973341
BC00476=973341
BC00477=887999
BC00478=846597
BC00479=930137
BC00480=969257
BC00481=969258
BC00482=969258
BC00483=999505
BC00484=999505
BC00485=999505
BC00486=999505
BC00487=999505
BC00488=999508
BC00489=999508
BC00490=999508
BC00491=973102
BC00492=973102
BC00493=904289
BC00494=812362
BC00495=476651
BC00496=522561
BC00497=566531
BC00498=593948
BC00499=593948
BC00500=529848
BC00501=529848
BC00502=333808
BC00503=333808
BC00504=333808
BC00505=294388
BC00506=294388
BC00507=461290
BC00508=663315
BC00509=778314
BC00510=778312
BC00511=778312
BC00512=778312
BC00513=838222
BC00514=838222
BC00515=566410
BC00516=679663
BC00517=656405
BC00518=656405
BC00519=717855
BC00520=717855
BC00521=717855
BC00522=662303
BC00523=657350
BC00524=657350
BC00525=718803
BC00526=718803
BC00527=717855
BC00528=792672
BC00529=792672
BC00530=896850
BC00531=895720
BC00532=895720
BC00533=957178
BC00534=957178
BC00535=978461
BC00536=957178
BC00537=792672
BC00538=792672
BC00539=792672
BC00540=887446
BC00541=903126
BC00542=903126
BC00543=903126
BC00544=964577
BC00545=976097
BC00546=993812
BC00547=964577
BC00548=887446
BC00549=792672
BC00550=792672
BC00551=700249
BC00552=546214
BC00553=546214
BC00554=546211
BC00555=546211
BC00556=406776
BC00557=406776
BC00558=406778
BC00559=468200
BC00560=468200
BC00561=546211
BC00562=546211
BC00563=546214
BC00564=546214
BC00565=507604
BC00566=410782
BC00567=410782
BC00568=410782
BC00569=472720
BC00570=472720
BC00571=507604
BC00572=546214
BC00573=546214
BC00574=516757
BC00575=383716
BC00576=349186
BC00577=349186
BC00578=336469
BC00579=349186
BC00580=410629
BC00581=416512
BC00582=515801
BC00583=520018
BC00584=474013
BC00585=474013
BC00586=403108
BC00587=336469
BC00588=349186
BC00589=349186
BC00590=349186
BC00591=337415
BC00592=337415
BC00593=336469
BC00594=336469
BC00595=428401
BC00596=546211
BC00597=591088
BC00598=591088
BC00599=591088
BC00600=531116
BC00601=529640
BC00602=529640
BC00603=529640
BC00604=529640
BC00605=546214
BC00606=589919
BC00607=595627
BC00608=595627
BC00609=534177
BC00610=534177
BC00611=546214
BC00612=529640
BC00613=651195
BC00614=765890
BC00615=777968
BC00616=778453
BC00617=779252
BC00618=840748
BC00619=840748
BC00620=765890
BC00621=717855
BC00622=741100
BC00623=780224
BC00624=780222
BC00625=841743
BC00626=841743
BC00627=741100
BC00628=717855
///POSTYPE BASE
///RECTAN
///RCONF 0,0,0,0,0,0,0,0,0,0,0,0,0,0,0,0,0,0,0,0,0,0,0,0
P00006=-2.449,0.031,8.825,0.0000,0.0000,0.0000
P00021=6.550,-0.003,-5.735,0.0000,0.0000,0.0000
P00022=5.943,-0.018,-6.388,0.0000,0.0000,0.0000
P00023=7.025,-0.019,-7.168,0.0000,0.0000,0.0000
P00024=5.926,-0.047,-4.777,0.0000,0.0000,0.0000
///RCONF 1,0,0,0,0,0,0,0,0,0,0,0,0,0,0,0,0,0,0,0,0,0,0,0
P00098=-0.089,-2.467,4.059,0.0000,0.0000,0.0000
P00099=0.011,-2.380,1.226,0.0000,0.0000,0.0000
P00100=-0.081,2.558,4.482,0.0000,0.0000,0.0000
P00101=0.030,-2.286,2.993,0.0000,0.0000,0.0000
P00102=-0.005,-1.108,1.644,0.0000,0.0000,0.0000
P00103=-0.094,-3.400,4.200,0.0000,0.0000,0.0000
P00104=0.043,-2.127,5.826,0.0000,0.0000,0.0000
P00105=-0.043,0.662,5.286,0.0000,0.0000,0.0000
P00106=-0.018,-2.519,0.237,0.0000,0.0000,0.0000
P00107=-0.008,-4.537,-4.500,0.0000,0.0000,0.0000
P00108=0.014,-3.040,2.637,0.0000,0.0000,0.0000
P00109=0.017,-3.622,2.341,0.0000,0.0000,0.0000
P00110=7346.140,158.997,-946.107,-0.1876,37.7131,-155.1643
P00111=7345.905,-141.160,-945.062,8.1413,34.2244,-174.1788
P00112=7393.287,158.977,-939.640,-0.1938,37.7128,-155.1905
P00113=7393.259,-141.170,-939.228,8.1507,34.2195,-174.1496
///RCONF 0,0,0,0,0,0,0,0,0,0,0,0,0,0,0,0,0,0,0,0,0,0,0,0
P00280=-0.761,-1.221,0.004,0.0000,0.0000,0.0000
///RCONF 1,0,0,0,0,0,0,0,0,0,0,0,0,0,0,0,0,0,0,0,0,0,0,0
P00281=-0.866,-3.587,-0.008,0.0000,0.0000,0.0000
///RCONF 0,0,0,0,1,0,0,0,0,0,0,0,0,0,0,0,0,0,0,0,0,0,0,0
P00290=-0.023,-0.050,5.560,0.0000,0.0000,0.0000
///RCONF 1,0,0,0,0,0,0,0,0,0,0,0,0,0,0,0,0,0,0,0,0,0,0,0
P00291=0.002,-0.893,4.526,0.0000,0.0000,0.0000
P00300=-0.036,-1.505,2.318,0.0000,0.0000,0.0000
///RCONF 0,0,0,0,0,0,0,0,0,0,0,0,0,0,0,0,0,0,0,0,0,0,0,0
P00301=0.005,-4.708,-4.628,0.0000,0.0000,0.0000
P00302=0.052,-2.937,-4.426,0.0000,0.0000,0.0000
P00303=-0.004,-1.437,-4.584,0.0000,0.0000,0.0000
P00304=0.028,-1.666,-4.234,0.0000,0.0000,0.0000
P00305=-0.003,-1.920,-3.501,0.0000,0.0000,0.0000
P00306=0.015,-2.252,-3.054,0.0000,0.0000,0.0000
P00307=0.019,-2.151,-5.077,0.0000,0.0000,0.0000
P00308=-0.003,-2.092,-4.888,0.0000,0.0000,0.0000
P00309=-0.040,-2.205,-4.992,0.0000,0.0000,0.0000
P00310=-0.006,-2.490,-5.925,0.0000,0.0000,0.0000
P00311=-0.007,-2.079,-5.307,0.0000,0.0000,0.0000
P00350=11.519,-0.008,1.149,0.0000,0.0000,0.0000
P00351=13.563,-0.027,-0.653,0.0000,0.0000,0.0000
P00352=13.252,-0.027,-0.827,0.0000,0.0000,0.0000
P00353=10.971,-0.082,0.776,0.0000,0.0000,0.0000
P00354=-0.024,2.508,-1.824,0.0000,0.0000,0.0000
P00355=-0.001,2.528,-1.131,0.0000,0.0000,0.0000
P00356=-0.034,2.921,-0.262,0.0000,0.0000,0.0000
P00357=0.003,3.386,-0.091,0.0000,0.0000,0.0000
P00358=0.014,3.037,-0.020,0.0000,0.0000,0.0000
P00359=-0.005,2.731,0.912,0.0000,0.0000,0.0000
P00360=-0.011,3.412,0.438,0.0000,0.0000,0.0000
P00361=0.018,3.050,1.253,0.0000,0.0000,0.0000
BP00110=5931.608
BP00111=5960.552
BP00112=5960.545
BP00113=5960.552
//INST
///DATE 2025/03/06 15:35
///ATTR SC,RW
///GROUP1 RB1,BS1
NOP
CALL JOB:MOVE_INTO_TUNNEL
MOVJ C00000 BC00000 VJ=30.00
'------------------------
'------------------------
'SPOINA SRODEK DOL
'------------------------
'------------------------
'POMIAR DO WYJ!! PRZEROBIC NA STD
MOVJ C00001 BC00001 VJ=40.00
MOVJ C00002 BC00002 VJ=40.00
'W3P
MOVJ C00003 BC00003 VJ=20.00 PL=0
MOVJ C00004 BC00004 VJ=20.00 PL=0
MOVL C00005 BC00005 V=166.7 PL=0
REFP 3 C00006 BC00006
CALL JOB:SEARCH-R1
SET P0099 P0006
SFTON P0099
MOVL C00007 BC00007 V=66.7 PL=0
REFP 3 C00008 BC00008
CALL JOB:SEARCH-R1
SET P0099 P0006
SFTON P0099
MOVL C00009 BC00009 V=333.3 PL=0
SFTOF
MOVJ C00010 BC00010 VJ=20.00 PL=0
MOVJ C00011 BC00011 VJ=20.00 PL=0
MOVL C00012 BC00012 V=166.7 PL=0
REFP 3 C00013 BC00013
CALL JOB:SEARCH-R1
SET P0098 P0006
SFTON P0098
MOVL C00014 BC00014 V=66.7 PL=0
REFP 3 C00015 BC00015
CALL JOB:SEARCH-R1
SET P0098 P0006
SFTON P0098
MOVL C00016 BC00016 V=333.3 PL=0
SFTOF
MOVJ C00017 BC00017 VJ=20.00 PL=0
MOVL C00018 BC00018 V=166.7 PL=0
REFP 3 C00019 BC00019
CALL JOB:SEARCH-R1
SET P0100 P0006
SFTON P0100
MOVL C00020 BC00020 V=66.7 PL=0
REFP 3 C00021 BC00021
CALL JOB:SEARCH-R1
SET P0100 P0006
SFTON P0100
MOVL C00022 BC00022 V=333.3 PL=0
SFTOF
'W3L
MOVL C00023 BC00023 V=666.7
MOVL C00024 BC00024 V=166.7 PL=0
REFP 3 C00025 BC00025
CALL JOB:SEARCH-R1
SET P0101 P0006
SFTON P0101
MOVL C00026 BC00026 V=166.7 PL=0
REFP 3 C00027 BC00027
CALL JOB:SEARCH-R1
SET P0101 P0006
SFTON P0101
MOVL C00028 BC00028 V=333.3 PL=0
SFTOF
'W9P
MOVL C00029 BC00029 V=666.7
MOVL C00030 BC00030 V=166.7
REFP 3 C00031 BC00031
CALL JOB:SEARCH-R1
SET P0102 P0006
SFTON P0102
MOVL C00032 BC00032 V=166.7 PL=0
REFP 3 C00033 BC00033
CALL JOB:SEARCH-R1
SET P0102 P0006
SFTON P0102
MOVL C00034 BC00034 V=333.3 PL=0
'W9L
MOVL C00035 BC00035 V=666.7
MOVL C00036 BC00036 V=166.7
REFP 3 C00037 BC00037
CALL JOB:SEARCH-R1
SET P0103 P0006
SFTON P0103
MOVL C00038 BC00038 V=166.7 PL=0
REFP 3 C00039 BC00039
CALL JOB:SEARCH-R1
SET P0103 P0006
SFTON P0103
MOVL C00040 BC00040 V=333.3 PL=0
'PRZEJAZ NAD BELKA
MOVL C00041 BC00041 V=666.7
MOVJ C00042 BC00042 VJ=40.00
MOVJ C00043 BC00043 VJ=40.00
MOVJ C00044 BC00044 VJ=40.00
'W1P
MOVJ C00045 BC00045 VJ=20.00 PL=0
MOVL C00046 BC00046 V=166.7 PL=0
REFP 3 C00047 BC00047
CALL JOB:SEARCH-R1
SET P0104 P0006
SFTON P0104
MOVL C00048 BC00048 V=166.7 PL=0
REFP 3 C00049 BC00049
CALL JOB:SEARCH-R1
SET P0104 P0006
SFTON P0104
MOVL C00050 BC00050 V=333.3 PL=0
SFTOF
'W1L
MOVL C00051 BC00051 V=666.7
MOVL C00052 BC00052 V=166.7 PL=0
REFP 3 C00053 BC00053
CALL JOB:SEARCH-R1
SET P0105 P0006
SFTON P0105
MOVL C00054 BC00054 V=166.7 PL=0
REFP 3 C00055 BC00055
CALL JOB:SEARCH-R1
SET P0105 P0006
SFTON P0105
MOVL C00056 BC00056 V=333.3 PL=0
SFTOF
MOVL C00057 BC00057 V=666.7
'W10P
MOVL C00058 BC00058 V=166.7 PL=0
REFP 3 C00059 BC00059
CALL JOB:SEARCH-R1
SET P0106 P0006
SFTON P0106
MOVL C00060 BC00060 V=166.7 PL=0
REFP 3 C00061 BC00061
CALL JOB:SEARCH-R1
SET P0106 P0006
SFTON P0106
MOVL C00062 BC00062 V=333.3 PL=0
SFTOF
'W10L
MOVL C00063 BC00063 V=333.3
MOVL C00064 BC00064 V=166.7 PL=0
REFP 3 C00065 BC00065
CALL JOB:SEARCH-R1
SET P0107 P0006
SFTON P0107
MOVL C00066 BC00066 V=166.7 PL=0
REFP 3 C00067 BC00067
CALL JOB:SEARCH-R1
SET P0107 P0006
SFTON P0107
MOVL C00068 BC00068 V=333.3 PL=0
SFTOF
MOVL C00069 BC00069 V=333.3
'PRZEJAZD
MOVJ C00070 BC00070 VJ=50.00
MOVJ C00071 BC00071 VJ=50.00
MOVJ C00072 BC00072 VJ=60.00
MOVJ C00073 BC00073 VJ=60.00
MOVJ C00074 BC00074 VJ=60.00
MOVJ C00075 BC00075 VJ=60.00 PL=0
MOVL C00076 BC00076 V=166.7 PL=0
REFP 3 C00077 BC00077
CALL JOB:SEARCH-R1
SET P0108 P0006
SFTON P0108
MOVL C00078 BC00078 V=166.7 PL=0
REFP 3 C00079 BC00079
CALL JOB:SEARCH-R1
SET P0108 P0006
SFTON P0108
MOVL C00080 BC00080 V=333.3 PL=0
SFTOF
'W2P
'W2L
MOVL C00081 BC00081 V=666.7
MOVL C00082 BC00082 V=166.7 PL=0
REFP 3 C00083 BC00083
CALL JOB:SEARCH-R1
SET P0109 P0006
SFTON P0109
MOVL C00084 BC00084 V=166.7 PL=0
REFP 3 C00085 BC00085
CALL JOB:SEARCH-R1
SET P0109 P0006
SFTON P0109
MOVL C00086 BC00086 V=333.3 PL=0
SFTOF
MOVJ C00087 BC00087 VJ=25.00
MOVJ C00088 BC00088 VJ=50.00
'W5L
MOVJ C00089 BC00089 VJ=30.00 PL=0
MOVL C00090 BC00090 V=166.7
REFP 3 C00091 BC00091
CALL JOB:SEARCH-R1
SET P0021 P0006
SFTON P0021
MOVL C00092 BC00092 V=166.7
REFP 3 C00093 BC00093
CALL JOB:SEARCH-R1
SET P0021 P0006
SFTON P0021
SFTOF
MOVL C00094 BC00094 V=166.7
'W6L
MOVJ C00095 BC00095 VJ=20.00 PL=0
MOVL C00096 BC00096 V=166.7
REFP 3 C00097 BC00097
CALL JOB:SEARCH-R1
SET P0022 P0006
SFTON P0022
MOVL C00098 BC00098 V=166.7
REFP 3 C00099 BC00099
CALL JOB:SEARCH-R1
SET P0022 P0006
SFTON P0022
SFTOF
MOVL C00100 BC00100 V=166.7
'W6P
MOVL C00101 BC00101 V=333.3 PL=0
REFP 3 C00102 BC00102
CALL JOB:SEARCH-R1
SET P0023 P0006
SFTON P0023
MOVL C00103 BC00103 V=166.7
REFP 3 C00104 BC00104
CALL JOB:SEARCH-R1
SET P0023 P0006
SFTON P0023
SFTOF
MOVL C00105 BC00105 V=166.7
'W5P
MOVJ C00106 BC00106 VJ=20.00 PL=0
MOVL C00107 BC00107 V=166.7
REFP 3 C00108 BC00108
CALL JOB:SEARCH-R1
SET P0024 P0006
SFTON P0024
MOVL C00109 BC00109 V=166.7
REFP 3 C00110 BC00110
CALL JOB:SEARCH-R1
SET P0024 P0006
SFTON P0024
SFTOF
MOVL C00111 BC00111 V=166.7
'W7A
MOVJ C00112 BC00112 VJ=40.00
MOVJ C00113 BC00113 VJ=40.00
MOVJ C00114 BC00114 VJ=40.00
MOVJ C00115 BC00115 VJ=40.00
MOVJ C00116 BC00116 VJ=40.00
MOVJ C00117 BC00117 VJ=40.00
MOVJ C00118 BC00118 VJ=40.00
MOVJ C00119 BC00119 VJ=40.00
MOVL C00120 BC00120 V=250.0
REFP 3 C00121 BC00121
CALL JOB:SEARCH-R1
SET P0280 P0006
SFTON P0280
MOVL C00122 BC00122 V=166.7
MOVL C00123 BC00123 V=250.0
MOVL C00124 BC00124 V=166.7
REFP 3 C00125 BC00125
CALL JOB:SEARCH-R1
SET P0280 P0006
MOVL C00126 BC00126 V=166.7
SFTOF
MOVL C00127 BC00127 V=333.3
MOVL C00128 BC00128 V=166.7
REFP 3 C00129 BC00129
CALL JOB:SEARCH-R1
SET P0290 P0006
SFTON P0290
MOVL C00130 BC00130 V=166.7
REFP 3 C00131 BC00131
CALL JOB:SEARCH-R1
SET P0290 P0006
MOVL C00132 BC00132 V=166.7
MOVJ C00133 BC00133 VJ=20.00
SFTOF
MOVJ C00134 BC00134 VJ=30.00
MOVJ C00135 BC00135 VJ=40.00
MOVJ C00136 BC00136 VJ=40.00
MOVJ C00137 BC00137 VJ=40.00
MOVJ C00138 BC00138 VJ=40.00
MOVJ C00139 BC00139 VJ=50.00
'W7B
MOVJ C00140 BC00140 VJ=50.00
MOVJ C00141 BC00141 VJ=50.00
MOVJ C00142 BC00142 VJ=30.00
MOVJ C00143 BC00143 VJ=20.00
MOVL C00144 BC00144 V=166.7
REFP 3 C00145 BC00145
CALL JOB:SEARCH-R1
SET P0281 P0006
MOVL C00146 BC00146 V=166.7
SFTON P0281
MOVL C00147 BC00147 V=166.7
MOVL C00148 BC00148 V=166.7
REFP 3 C00149 BC00149
CALL JOB:SEARCH-R1
SET P0281 P0006
MOVJ C00150 BC00150 VJ=15.00
SFTOF
MOVJ C00151 BC00151 VJ=20.00
MOVL C00152 BC00152 V=166.7
REFP 3 C00153 BC00153
CALL JOB:SEARCH-R1
SET P0291 P0006
MOVL C00154 BC00154 V=166.7
MOVL C00155 BC00155 V=166.7
REFP 3 C00156 BC00156
CALL JOB:SEARCH-R1
SET P0291 P0006
MOVL C00157 BC00157 V=166.7
COMM MOVJ C00158 BC00158 VJ=40.00
COMM MOVJ C00159 BC00159 VJ=50.00
COMM 'W5L
COMM MOVJ C00160 BC00160 VJ=30.00 PL=0
COMM SET I020 110
COMM CALL JOB:SEARCH_Z-40_Z1_X40
COMM MOVL C00161 BC00161 V=166.7
COMM 'W6L
COMM MOVJ C00162 BC00162 VJ=20.00 PL=0
COMM SET I020 112
COMM CALL JOB:SEARCH_Z-40_Z1_X40
COMM MOVL C00163 BC00163 V=166.7
COMM 'W6P
COMM MOVL C00164 BC00164 V=150.0 PL=0
COMM SET I020 113
COMM CALL JOB:SEARCH_Z-40_Z1_X40
COMM MOVL C00165 BC00165 V=166.7
COMM 'W5P
COMM MOVJ C00166 BC00166 VJ=20.00 PL=0
COMM SET I020 111
COMM CALL JOB:SEARCH_Z-40_Z1_X40
COMM MOVL C00167 BC00167 V=166.7
COMM 'W7A
COMM MOVJ C00168 BC00168 VJ=40.00
COMM MOVJ C00169 BC00169 VJ=40.00
COMM MOVJ C00170 BC00170 VJ=40.00
COMM MOVJ C00171 BC00171 VJ=40.00
COMM MOVJ C00172 BC00172 VJ=40.00
COMM MOVJ C00173 BC00173 VJ=40.00
COMM MOVJ C00174 BC00174 VJ=40.00
COMM MOVJ C00175 BC00175 VJ=40.00
COMM MOVL C00176 BC00176 V=250.0
COMM REFP 3 C00177 BC00177
COMM CALL JOB:SEARCH-R1
COMM SET P0280 P0006
COMM SFTON P0280
COMM MOVL C00178 BC00178 V=166.7
COMM MOVL C00179 BC00179 V=250.0
COMM MOVL C00180 BC00180 V=166.7
COMM REFP 3 C00181 BC00181
COMM CALL JOB:SEARCH-R1
COMM SET P0280 P0006
COMM MOVL C00182 BC00182 V=166.7
COMM SFTOF
COMM MOVL C00183 BC00183 V=333.3
COMM MOVL C00184 BC00184 V=166.7
COMM REFP 3 C00185 BC00185
COMM CALL JOB:SEARCH-R1
COMM SET P0290 P0006
COMM SFTON P0290
COMM MOVL C00186 BC00186 V=166.7
COMM REFP 3 C00187 BC00187
COMM CALL JOB:SEARCH-R1
COMM SET P0290 P0006
COMM MOVL C00188 BC00188 V=166.7
COMM 'DOKONCZYC SEARCH
COMM 'DOKONCZYC SEARCH
COMM MOVJ C00189 BC00189 VJ=20.00
COMM SFTOF
COMM MOVJ C00190 BC00190 VJ=30.00
COMM MOVJ C00191 BC00191 VJ=40.00
COMM MOVJ C00192 BC00192 VJ=40.00
COMM MOVJ C00193 BC00193 VJ=40.00
COMM MOVJ C00194 BC00194 VJ=40.00
COMM MOVJ C00195 BC00195 VJ=50.00
COMM 'W7B
COMM MOVJ C00196 BC00196 VJ=50.00
COMM MOVJ C00197 BC00197 VJ=50.00
COMM MOVJ C00198 BC00198 VJ=30.00
COMM MOVJ C00199 BC00199 VJ=20.00
COMM MOVL C00200 BC00200 V=166.7
COMM REFP 3 C00201 BC00201
COMM CALL JOB:SEARCH-R1
COMM SET P0281 P0006
COMM MOVL C00202 BC00202 V=166.7
COMM SFTON P0281
COMM MOVL C00203 BC00203 V=166.7
COMM MOVL C00204 BC00204 V=166.7
COMM REFP 3 C00205 BC00205
COMM CALL JOB:SEARCH-R1
COMM SET P0281 P0006
COMM MOVJ C00206 BC00206 VJ=15.00
COMM SFTOF
COMM MOVJ C00207 BC00207 VJ=20.00
COMM MOVL C00208 BC00208 V=166.7
COMM REFP 3 C00209 BC00209
COMM CALL JOB:SEARCH-R1
COMM SET P0291 P0006
COMM MOVL C00210 BC00210 V=166.7
COMM MOVL C00211 BC00211 V=166.7
COMM REFP 3 C00212 BC00212
COMM CALL JOB:SEARCH-R1
COMM SET P0291 P0006
COMM MOVL C00213 BC00213 V=166.7
COMM 'DOKONCZYC SEARCH
COMM 'DOKONCZYC SEARCH
COMM 'DOKONCZYC SEARCH
MOVJ C00214 BC00214 VJ=30.00
MOVJ C00215 BC00215 VJ=30.00
MOVJ C00216 BC00216 VJ=50.00
MOVJ C00217 BC00217 VJ=50.00
'------------------------
'------------------------
'PRAWA STRONA PROFIL GORA
'------------------------
'------------------------
MOVJ C00218 BC00218 VJ=50.00
MOVJ C00219 BC00219 VJ=50.00
MOVJ C00220 BC00220 VJ=50.00
MOVJ C00221 BC00221 VJ=20.00
MOVJ C00222 BC00222 VJ=50.00
'------------------------
'W14A L
'------------------------
SFTOF
MOVJ C00223 BC00223 VJ=50.00
MOVJ C00224 BC00224 VJ=30.00
MOVL C00225 BC00225 V=166.7 PL=0
REFP 3 C00226 BC00226
CALL JOB:SEARCH-R1
SET P0300 P0006
SFTON P0300
MOVL C00227 BC00227 V=166.7 PL=0
REFP 3 C00228 BC00228
CALL JOB:SEARCH-R1
SET P0300 P0006
SFTON P0300
MOVL C00229 BC00229 V=166.7 PL=0
SFTOF
'------------------------
'W14A P
'------------------------
SFTOF
MOVJ C00230 BC00230 VJ=50.00
MOVJ C00231 BC00231 VJ=50.00
MOVL C00232 BC00232 V=166.7 PL=0
REFP 3 C00233 BC00233
CALL JOB:SEARCH-R1
SET P0301 P0006
SFTON P0301
MOVL C00234 BC00234 V=166.7 PL=0
REFP 3 C00235 BC00235
CALL JOB:SEARCH-R1
SET P0301 P0006
SFTON P0301
MOVL C00236 BC00236 V=166.7 PL=0
SFTOF
'------------------------
'W19A L
'------------------------
SFTOF
MOVJ C00237 BC00237 VJ=50.00
MOVL C00238 BC00238 V=200.0 PL=0
REFP 3 C00239 BC00239
CALL JOB:SEARCH-R1
SET P0302 P0006
SFTON P0302
MOVL C00240 BC00240 V=166.7 PL=0
REFP 3 C00241 BC00241
CALL JOB:SEARCH-R1
SET P0302 P0006
SFTON P0302
MOVL C00242 BC00242 V=250.0 PL=0
SFTOF
'------------------------
'W19A P
'------------------------
SFTOF
MOVJ C00243 BC00243 VJ=50.00
MOVL C00244 BC00244 V=166.7 PL=0
REFP 3 C00245 BC00245
CALL JOB:SEARCH-R1
SET P0303 P0006
SFTON P0303
MOVL C00246 BC00246 V=166.7 PL=0
REFP 3 C00247 BC00247
CALL JOB:SEARCH-R1
SET P0303 P0006
SFTON P0303
MOVL C00248 BC00248 V=166.7 PL=0
SFTOF
'------------------------
'W13A L
'------------------------
SFTOF
MOVJ C00249 BC00249 VJ=50.00
MOVL C00250 BC00250 V=166.7 PL=0
REFP 3 C00251 BC00251
CALL JOB:SEARCH-R1
SET P0304 P0006
SFTON P0304
MOVL C00252 BC00252 V=166.7 PL=0
REFP 3 C00253 BC00253
CALL JOB:SEARCH-R1
SET P0304 P0006
SFTON P0304
MOVL C00254 BC00254 V=166.7 PL=0
SFTOF
'------------------------
'W13A P
'------------------------
SFTOF
MOVJ C00255 BC00255 VJ=50.00
MOVL C00256 BC00256 V=200.0 PL=0
REFP 3 C00257 BC00257
CALL JOB:SEARCH-R1
SET P0305 P0006
SFTON P0305
MOVL C00258 BC00258 V=166.7 PL=0
REFP 3 C00259 BC00259
CALL JOB:SEARCH-R1
SET P0305 P0006
SFTON P0305
MOVL C00260 BC00260 V=250.0 PL=0
SFTOF
'------------------------
'W18A L
'------------------------
SFTOF
MOVJ C00261 BC00261 VJ=50.00
MOVL C00262 BC00262 V=200.0 PL=0
REFP 3 C00263 BC00263
CALL JOB:SEARCH-R1
SET P0306 P0006
SFTON P0306
MOVL C00264 BC00264 V=166.7 PL=0
REFP 3 C00265 BC00265
CALL JOB:SEARCH-R1
SET P0306 P0006
SFTON P0306
MOVL C00266 BC00266 V=166.7 PL=0
SFTOF
'------------------------
'W18A P
'------------------------
SFTOF
MOVJ C00267 BC00267 VJ=50.00
MOVL C00268 BC00268 V=200.0 PL=0
REFP 3 C00269 BC00269
CALL JOB:SEARCH-R1
SET P0307 P0006
SFTON P0307
MOVL C00270 BC00270 V=166.7 PL=0
REFP 3 C00271 BC00271
CALL JOB:SEARCH-R1
SET P0307 P0006
SFTON P0307
MOVL C00272 BC00272 V=166.7 PL=0
SFTOF
'------------------------
'W15A L
'------------------------
SFTOF
MOVJ C00273 BC00273 VJ=50.00
MOVL C00274 BC00274 V=200.0 PL=0
REFP 3 C00275 BC00275
CALL JOB:SEARCH-R1
SET P0308 P0006
SFTON P0308
MOVL C00276 BC00276 V=166.7 PL=0
REFP 3 C00277 BC00277
CALL JOB:SEARCH-R1
SET P0308 P0006
SFTON P0308
MOVL C00278 BC00278 V=166.7 PL=0
SFTOF
'------------------------
'W15A P
'------------------------
SFTOF
MOVJ C00279 BC00279 VJ=50.00
MOVL C00280 BC00280 V=166.7 PL=0
REFP 3 C00281 BC00281
CALL JOB:SEARCH-R1
SET P0309 P0006
SFTON P0309
MOVL C00282 BC00282 V=166.7 PL=0
REFP 3 C00283 BC00283
CALL JOB:SEARCH-R1
SET P0309 P0006
SFTON P0309
MOVL C00284 BC00284 V=166.7 PL=0
SFTOF
MOVL C00285 BC00285 V=333.3
'------------------------
'W17A L
'------------------------
MOVL C00286 BC00286 V=500.0
SFTOF
MOVJ C00287 BC00287 VJ=20.00
MOVL C00288 BC00288 V=166.7 PL=0
REFP 3 C00289 BC00289
CALL JOB:SEARCH-R1
SET P0310 P0006
SFTON P0310
MOVL C00290 BC00290 V=166.7 PL=0
REFP 3 C00291 BC00291
CALL JOB:SEARCH-R1
SET P0310 P0006
SFTON P0310
MOVL C00292 BC00292 V=166.7 PL=0
SFTOF
'------------------------
'W17A P
'------------------------
SFTOF
MOVL C00293 BC00293 V=416.7
MOVL C00294 BC00294 V=166.7 PL=0
REFP 3 C00295 BC00295
CALL JOB:SEARCH-R1
SET P0311 P0006
SFTON P0311
MOVL C00296 BC00296 V=166.7 PL=0
REFP 3 C00297 BC00297
CALL JOB:SEARCH-R1
SET P0311 P0006
SFTON P0311
MOVL C00298 BC00298 V=166.7 PL=0
SFTOF
MOVJ C00299 BC00299 VJ=10.00
MOVJ C00300 BC00300 VJ=20.00
MOVJ C00301 BC00301 VJ=50.00
MOVJ C00302 BC00302 VJ=50.00
MOVJ C00303 BC00303 VJ=70.00
MOVJ C00304 BC00304 VJ=30.00
MOVJ C00305 BC00305 VJ=30.00
'------------------------
'------------------------
'LEWA STRONA PROFIL GORA
'------------------------
'------------------------
MOVJ C00306 BC00306 VJ=30.00
MOVJ C00307 BC00307 VJ=30.00
MOVJ C00308 BC00308 VJ=30.00
'------------------------
'W17B L
'------------------------
SFTOF
MOVJ C00309 BC00309 VJ=15.00
MOVL C00310 BC00310 V=166.7 PL=0
REFP 3 C00311 BC00311
CALL JOB:SEARCH-R1
SET P0350 P0006
SFTON P0350
MOVL C00312 BC00312 V=166.7 PL=0
REFP 3 C00313 BC00313
CALL JOB:SEARCH-R1
SET P0350 P0006
SFTON P0350
MOVL C00314 BC00314 V=166.7 PL=0
SFTOF
'------------------------
'W17B P
'------------------------
SFTOF
MOVL C00315 BC00315 V=333.3
MOVL C00316 BC00316 V=166.7 PL=0
REFP 3 C00317 BC00317
CALL JOB:SEARCH-R1
SET P0351 P0006
SFTON P0351
MOVL C00318 BC00318 V=166.7 PL=0
REFP 3 C00319 BC00319
CALL JOB:SEARCH-R1
SET P0351 P0006
SFTON P0351
MOVL C00320 BC00320 V=166.7 PL=0
SFTOF
'POPRAWID DOJAZD
'------------------------
'W15B L
'------------------------
SFTOF
MOVJ C00321 BC00321 VJ=10.00
MOVL C00322 BC00322 V=166.7 PL=0
REFP 3 C00323 BC00323
CALL JOB:SEARCH-R1
SET P0352 P0006
SFTON P0352
MOVL C00324 BC00324 V=166.7 PL=0
REFP 3 C00325 BC00325
CALL JOB:SEARCH-R1
SET P0352 P0006
SFTON P0352
MOVL C00326 BC00326 V=166.7 PL=0
SFTOF
'------------------------
'W15B P
'------------------------
SFTOF
MOVJ C00327 BC00327 VJ=20.00
MOVL C00328 BC00328 V=166.7 PL=0
REFP 3 C00329 BC00329
CALL JOB:SEARCH-R1
SET P0353 P0006
SFTON P0353
MOVL C00330 BC00330 V=166.7 PL=0
REFP 3 C00331 BC00331
CALL JOB:SEARCH-R1
SET P0353 P0006
SFTON P0353
MOVL C00332 BC00332 V=166.7 PL=0
SFTOF
'------------------------
'W18B L
'------------------------
SFTOF
MOVJ C00333 BC00333 VJ=50.00
MOVL C00334 BC00334 V=166.7 PL=0
REFP 3 C00335 BC00335
CALL JOB:SEARCH-R1
SET P0354 P0006
SFTON P0354
MOVL C00336 BC00336 V=166.7 PL=0
REFP 3 C00337 BC00337
CALL JOB:SEARCH-R1
SET P0354 P0006
SFTON P0354
MOVL C00338 BC00338 V=166.7 PL=0
SFTOF
'------------------------
'W18B P
'------------------------
SFTOF
MOVJ C00339 BC00339 VJ=50.00
MOVL C00340 BC00340 V=166.7 PL=0
REFP 3 C00341 BC00341
CALL JOB:SEARCH-R1
SET P0355 P0006
SFTON P0355
MOVL C00342 BC00342 V=166.7 PL=0
REFP 3 C00343 BC00343
CALL JOB:SEARCH-R1
SET P0355 P0006
SFTON P0355
MOVL C00344 BC00344 V=166.7 PL=0
SFTOF
'------------------------
'W13B L
'------------------------
SFTOF
MOVJ C00345 BC00345 VJ=50.00
MOVL C00346 BC00346 V=166.7 PL=0
REFP 3 C00347 BC00347
CALL JOB:SEARCH-R1
SET P0356 P0006
SFTON P0356
MOVL C00348 BC00348 V=166.7 PL=0
REFP 3 C00349 BC00349
CALL JOB:SEARCH-R1
SET P0356 P0006
SFTON P0356
MOVL C00350 BC00350 V=166.7 PL=0
SFTOF
'------------------------
'W13B P
'------------------------
SFTOF
MOVJ C00351 BC00351 VJ=50.00
MOVL C00352 BC00352 V=166.7 PL=0
REFP 3 C00353 BC00353
CALL JOB:SEARCH-R1
SET P0357 P0006
SFTON P0357
MOVL C00354 BC00354 V=166.7 PL=0
REFP 3 C00355 BC00355
CALL JOB:SEARCH-R1
SET P0357 P0006
SFTON P0357
MOVL C00356 BC00356 V=166.7 PL=0
SFTOF
'------------------------
'W19B L
'------------------------
SFTOF
MOVJ C00357 BC00357 VJ=50.00
MOVL C00358 BC00358 V=166.7 PL=0
REFP 3 C00359 BC00359
CALL JOB:SEARCH-R1
SET P0358 P0006
SFTON P0358
MOVL C00360 BC00360 V=166.7 PL=0
REFP 3 C00361 BC00361
CALL JOB:SEARCH-R1
SET P0358 P0006
SFTON P0358
MOVL C00362 BC00362 V=166.7 PL=0
SFTOF
'------------------------
'W19B P
'------------------------
SFTOF
MOVJ C00363 BC00363 VJ=50.00
MOVL C00364 BC00364 V=166.7 PL=0
REFP 3 C00365 BC00365
CALL JOB:SEARCH-R1
SET P0359 P0006
SFTON P0359
MOVL C00366 BC00366 V=166.7 PL=0
REFP 3 C00367 BC00367
CALL JOB:SEARCH-R1
SET P0359 P0006
SFTON P0359
MOVL C00368 BC00368 V=166.7 PL=0
SFTOF
'------------------------
'W14B L
'------------------------
SFTOF
MOVJ C00369 BC00369 VJ=50.00
MOVL C00370 BC00370 V=166.7 PL=0
REFP 3 C00371 BC00371
CALL JOB:SEARCH-R1
SET P0360 P0006
SFTON P0360
MOVL C00372 BC00372 V=166.7 PL=0
REFP 3 C00373 BC00373
CALL JOB:SEARCH-R1
SET P0360 P0006
SFTON P0360
MOVL C00374 BC00374 V=166.7 PL=0
SFTOF
'------------------------
'W14B P
'------------------------
SFTOF
MOVJ C00375 BC00375 VJ=50.00
MOVL C00376 BC00376 V=166.7 PL=0
REFP 3 C00377 BC00377
CALL JOB:SEARCH-R1
SET P0361 P0006
SFTON P0361
MOVL C00378 BC00378 V=166.7 PL=0
REFP 3 C00379 BC00379
CALL JOB:SEARCH-R1
SET P0361 P0006
SFTON P0361
MOVL C00380 BC00380 V=166.7 PL=0
SFTOF
MOVJ C00381 BC00381 VJ=50.00
MOVJ C00382 BC00382 VJ=50.00
MOVJ C00383 BC00383 VJ=50.00
MOVJ C00384 BC00384 VJ=50.00
'WELD
'WELD
'WELD
MOVJ C00385 BC00385 VJ=10.00
'**********************
'**********************
'POCZATEK SPAWANIA DOL
'**********************
'**********************
''
'**********************
'W1
'**********************
MOVJ C00386 BC00386 VJ=50.00
MOVJ C00387 BC00387 VJ=40.00
MOVL C00388 BC00388 V=166.7
SFTON P0104
MOVL C00389 BC00389 V=166.7
MACRO1 MJ#(0) ARGF24
ARCON
SFTON P0105
MOVL C00390 BC00390 V=11.7
ARCOF
SFTOF
MOVJ C00391 BC00391 VJ=20.00
MOVJ C00392 BC00392 VJ=30.00
MOVJ C00393 BC00393 VJ=50.00
MOVJ C00394 BC00394 VJ=40.00
MOVJ C00395 BC00395 VJ=20.00
'**********************
'W2
'**********************
SFTON P0108
MOVL C00396 BC00396 V=166.7 PL=0
ARCON
SFTON P0109
MOVL C00397 BC00397 V=11.7
MOVL C00398 BC00398 V=11.7
ARCOF
SFTOF
MOVL C00399 BC00399 V=333.3
MOVJ C00400 BC00400 VJ=40.00
MOVJ C00401 BC00401 VJ=70.00
MOVJ C00402 BC00402 VJ=20.00
MOVL C00403 BC00403 V=666.7
'**********************
'W3
'**********************
SFTON P0101
MOVL C00404 BC00404 V=166.7
ARCON
SFTON P0100
MOVL C00405 BC00405 V=11.7
ARCOF
MOVL C00406 BC00406 V=166.7
SFTOF
MOVJ C00407 BC00407 VJ=30.00
MOVJ C00408 BC00408 VJ=30.00
MOVJ C00409 BC00409 VJ=50.00
MOVJ C00410 BC00410 VJ=30.00
MOVJ C00411 BC00411 VJ=40.00
'**********************
'W5
'**********************
MOVJ C00412 BC00412 VJ=50.00
MOVJ C00413 BC00413 VJ=25.00
MOVJ C00414 BC00414 VJ=30.00
MOVL C00415 BC00415 V=333.3
'**********************
MACRO1 MJ#(0) ARGF9
SFTON P0024
MOVL C00416 BC00416 V=166.7
ARCON
WVON WEV#(2)
SFTON P0021
MOVL C00417 BC00417 V=10.8
ARCOF
WVOF
SFTOF
MOVJ C00418 BC00418 VJ=20.00
MOVJ C00419 BC00419 VJ=20.00
'**********************
'W6
'**********************
MACRO1 MJ#(0) ARGF9
SFTON P0023
MOVL C00420 BC00420 V=250.0
ARCON
WVON WEV#(2)
SFTON P0022
MOVL C00421 BC00421 V=10.8
ARCOF
WVOF
SFTOF
MOVJ C00422 BC00422 VJ=10.00
MOVJ C00423 BC00423 VJ=30.00
MOVJ C00424 BC00424 VJ=40.00
MOVJ C00425 BC00425 VJ=40.00
MOVJ C00426 BC00426 VJ=40.00
MOVJ C00427 BC00427 VJ=40.00
MOVJ C00428 BC00428 VJ=20.00
MOVJ C00429 BC00429 VJ=10.00
MOVJ C00430 BC00430 VJ=20.00
MOVL C00431 BC00431 V=166.7
MACRO1 MJ#(0) ARGF14
MOVL C00432 BC00432 V=166.7
SFTON P0280
MOVL C00433 BC00433 V=166.7 PL=0
ARCON ASF#(22)
MOVL C00434 BC00434 V=9.2
MOVL C00435 BC00435 V=9.2
SFTON P0290
MOVL C00436 BC00436 V=9.2
MOVL C00437 BC00437 V=9.2
ARCOF
SFTOF
MOVL C00438 BC00438 V=250.0
MOVL C00439 BC00439 V=416.7
MOVJ C00440 BC00440 VJ=30.00
MOVJ C00441 BC00441 VJ=30.00
MOVJ C00442 BC00442 VJ=30.00
MOVJ C00443 BC00443 VJ=30.00
MOVJ C00444 BC00444 VJ=30.00
'7b
MOVL C00445 BC00445 V=333.3
MOVL C00446 BC00446 V=333.3
SFTON P0281
MOVL C00447 BC00447 V=166.7 PL=0
ARCON ASF#(22)
MOVL C00448 BC00448 V=9.2
MOVL C00449 BC00449 V=9.2
SFTON P0291
MOVL C00450 BC00450 V=9.2
MOVL C00451 BC00451 V=9.2
MOVL C00452 BC00452 V=9.2
ARCOF
SFTOF
'TUTAJ DODAC 7
'TUTAJ DODAC 7
'TUTAJ DODAC 7
MOVL C00453 BC00453 V=333.3
MOVL C00454 BC00454 V=333.3
MOVL C00455 BC00455 V=333.3
COMM '**********************
COMM 'W5
COMM '**********************
COMM MACRO1 MJ#(0) ARGF9
COMM SFTON P0021
COMM MOVL P0111 BP111 V=66.7
COMM ARCON
COMM MOVL P0110 BP110 V=10.0
COMM ARCOF
COMM SFTOF
COMM MOVJ C00456 BC00456 VJ=20.00
COMM MOVJ C00457 BC00457 VJ=20.00
COMM '**********************
COMM 'W6
COMM '**********************
COMM MACRO1 MJ#(0) ARGF9
COMM SFTON P0023
COMM MOVL P0113 BP113 V=66.7
COMM ARCON
COMM MOVL P0112 BP112 V=10.8
COMM ARCOF
COMM SFTOF
COMM MOVJ C00458 BC00458 VJ=10.00
COMM MOVJ C00459 BC00459 VJ=30.00
COMM MOVJ C00460 BC00460 VJ=30.00
COMM MOVJ C00461 BC00461 VJ=40.00
COMM MOVJ C00462 BC00462 VJ=40.00
COMM MOVJ C00463 BC00463 VJ=40.00
COMM MOVJ C00464 BC00464 VJ=40.00
COMM MOVJ C00465 BC00465 VJ=20.00
COMM MOVJ C00466 BC00466 VJ=10.00
COMM MOVJ C00467 BC00467 VJ=20.00
COMM MOVL C00468 BC00468 V=166.7
COMM MACRO1 MJ#(0) ARGF14
COMM MOVL C00469 BC00469 V=166.7
COMM SFTON P0280
COMM MOVL C00470 BC00470 V=166.7 PL=0
COMM ARCON ASF#(22)
COMM MOVL C00471 BC00471 V=9.2
COMM MOVL C00472 BC00472 V=9.2
COMM SFTON P0281
COMM MOVL C00473 BC00473 V=9.2
COMM MOVL C00474 BC00474 V=9.2
COMM ARCOF
COMM SFTOF
COMM MOVL C00475 BC00475 V=250.0
COMM MOVL C00476 BC00476 V=416.7
COMM MOVJ C00477 BC00477 VJ=30.00
COMM MOVJ C00478 BC00478 VJ=30.00
COMM MOVJ C00479 BC00479 VJ=30.00
COMM MOVJ C00480 BC00480 VJ=30.00
COMM MOVJ C00481 BC00481 VJ=30.00
COMM '7b
COMM MOVL C00482 BC00482 V=333.3
COMM MOVL C00483 BC00483 V=333.3
COMM SFTON P0281
COMM MOVL C00484 BC00484 V=166.7 PL=0
COMM ARCON ASF#(22)
COMM MOVL C00485 BC00485 V=9.2
COMM MOVL C00486 BC00486 V=9.2
COMM SFTON P0291
COMM MOVL C00487 BC00487 V=9.2
COMM MOVL C00488 BC00488 V=9.2
COMM MOVL C00489 BC00489 V=9.2
COMM ARCOF
COMM SFTOF
COMM 'TUTAJ DODAC 7
COMM 'TUTAJ DODAC 7
COMM 'TUTAJ DODAC 7
COMM MOVL C00490 BC00490 V=333.3
COMM MOVL C00491 BC00491 V=333.3
COMM MOVL C00492 BC00492 V=333.3
MOVJ C00493 BC00493 VJ=20.00
MOVJ C00494 BC00494 VJ=30.00
MOVJ C00495 BC00495 VJ=50.00
MOVJ C00496 BC00496 VJ=50.00
MOVJ C00497 BC00497 VJ=40.00
MOVJ C00498 BC00498 VJ=10.00
'**********************
'W9
'**********************
SFTON P0103
MACRO1 MJ#(0) ARGF24
MOVL C00499 BC00499 V=166.7
ARCON
SFTON P0102
MOVL C00500 BC00500 V=11.7
ARCOF
SFTOF
MOVL C00501 BC00501 V=166.7
'dod spoina podloga(bez rozpurek)
MOVL C00502 BC00502 V=666.7
'**********************
'....
'**********************
MOVL C00503 BC00503 V=666.7
SFTON P0098
MOVL C00504 BC00504 V=166.7 PL=0
ARCON
SFTON P0099
MOVL C00505 BC00505 V=11.7
ARCOF
MOVL C00506 BC00506 V=166.7
SFTOF
MOVJ C00507 BC00507 VJ=40.00
MOVJ C00508 BC00508 VJ=70.00
MOVJ C00509 BC00509 VJ=50.00
MOVJ C00510 BC00510 VJ=20.00
'**********************
'W10
'**********************
MOVL C00511 BC00511 V=333.3
SFTON P0106
MOVL C00512 BC00512 V=166.7
ARCON
SFTON P0107
MOVL C00513 BC00513 V=11.7
ARCOF
SFTOF
MOVL C00514 BC00514 V=333.3
MOVJ C00515 BC00515 VJ=50.00
'**********************
'**********************
'POCZATEK SPAWANIA BOKI
'**********************
'**********************
MOVJ C00516 BC00516 VJ=50.00
MOVJ C00517 BC00517 VJ=50.00
'**********************
'W13A
'**********************
SFTON P0305
MOVL C00518 BC00518 V=250.0 PL=0
SFTOF
MACRO1 MJ#(0) ARGF10
ARCON
SFTON P0304
MOVL C00519 BC00519 V=10.8
ARCOF
SFTOF
MOVL C00520 BC00520 V=250.0
'W13B
MOVJ C00521 BC00521 VJ=30.00
MOVJ C00522 BC00522 VJ=50.00
MOVL C00523 BC00523 V=500.0
'**********************
'W13B
'**********************
SFTON P0356
MOVL C00524 BC00524 V=133.3 PL=0
SFTOF
ARCON
SFTON P0357
MOVL C00525 BC00525 V=10.8
ARCOF
SFTOF
MOVL C00526 BC00526 V=250.0
MOVJ C00527 BC00527 VJ=30.00
MOVJ C00528 BC00528 VJ=40.00
MOVJ C00529 BC00529 VJ=30.00
MOVJ C00530 BC00530 VJ=30.00
'**********************
'W14A
'**********************
MOVL C00531 BC00531 V=250.0
SFTON P0301
MOVL C00532 BC00532 V=50.0 PL=0
SFTOF
ARCON
SFTON P0300
MOVL C00533 BC00533 V=10.8
MOVL C00534 BC00534 V=10.8
MOVL C00535 BC00535 V=10.8
ARCOF
SFTOF
MOVL C00536 BC00536 V=150.0
MOVJ C00537 BC00537 VJ=40.00
MOVJ C00538 BC00538 VJ=30.00
MOVJ C00539 BC00539 VJ=30.00
MOVJ C00540 BC00540 VJ=30.00
MOVJ C00541 BC00541 VJ=30.00
'**********************
'W14B
'**********************
SFTON P0360
MOVL C00542 BC00542 V=333.3
MOVL C00543 BC00543 V=166.7 PL=0
SFTOF
ARCON
SFTON P0361
MOVL C00544 BC00544 V=10.8
MOVL C00545 BC00545 V=10.8
MOVL C00546 BC00546 V=10.8
ARCOF
SFTOF
MOVL C00547 BC00547 V=250.0
MOVJ C00548 BC00548 VJ=40.00
MOVJ C00549 BC00549 VJ=40.00
MOVJ C00550 BC00550 VJ=30.00
MOVJ C00551 BC00551 VJ=40.00
MOVJ C00552 BC00552 VJ=30.00
MOVJ C00553 BC00553 VJ=30.00
MOVJ C00554 BC00554 VJ=30.00
MOVJ C00555 BC00555 VJ=30.00
MOVJ C00556 BC00556 VJ=30.00
'**********************
'W15A
'**********************
SFTON P0309
MOVL C00557 BC00557 V=166.7
MOVL C00558 BC00558 V=166.7 PL=0
SFTOF
ARCON
SFTON P0308
MOVL C00559 BC00559 V=10.8
ARCOF
SFTOF
MOVL C00560 BC00560 V=150.0
MOVJ C00561 BC00561 VJ=30.00
MOVJ C00562 BC00562 VJ=50.00
MOVJ C00563 BC00563 VJ=50.00
MOVJ C00564 BC00564 VJ=50.00
MOVJ C00565 BC00565 VJ=50.00
MOVJ C00566 BC00566 VJ=50.00
'**********************
'W15B
'**********************
SFTON P0352
MOVL C00567 BC00567 V=250.0
MOVL C00568 BC00568 V=83.3 PL=0
SFTOF
ARCON
SFTON P0353
MOVL C00569 BC00569 V=10.8
ARCOF
MOVL C00570 BC00570 V=66.7
SFTOF
MOVJ C00571 BC00571 VJ=40.00
MOVJ C00572 BC00572 VJ=50.00
MOVJ C00573 BC00573 VJ=50.00
'BRAK W TEJ DLUGOSCI
'**********************
'W16A
'**********************
'**********************
'W16B
'**********************
'BRAK W TEJ DLUGOSCI
'**********************
'W17A
'**********************
MOVJ C00574 BC00574 VJ=50.00
MOVJ C00575 BC00575 VJ=50.00
'**********************
'W17A
'**********************
SFTON P0310
MOVL C00576 BC00576 V=333.3
MOVL C00577 BC00577 V=166.7 PL=0
SFTOF
ARCON
SFTON P0311
MOVL C00578 BC00578 V=10.8
ARCOF
SFTOF
MOVL C00579 BC00579 V=333.3
MOVJ C00580 BC00580 VJ=30.00
MOVJ C00581 BC00581 VJ=30.00
MOVJ C00582 BC00582 VJ=50.00
MOVJ C00583 BC00583 VJ=50.00
MOVJ C00584 BC00584 VJ=50.00
MOVJ C00585 BC00585 VJ=50.00
MOVJ C00586 BC00586 VJ=50.00
MOVJ C00587 BC00587 VJ=30.00
MOVJ C00588 BC00588 VJ=30.00
'**********************
'W17B
'**********************
SFTON P0351
MOVL C00589 BC00589 V=166.7
MOVL C00590 BC00590 V=166.7 PL=0
SFTOF
ARCON
SFTON P0350
MOVL C00591 BC00591 V=10.8
ARCOF
SFTOF
MOVL C00592 BC00592 V=250.0
MOVJ C00593 BC00593 VJ=30.00
MOVJ C00594 BC00594 VJ=30.00
MOVJ C00595 BC00595 VJ=30.00
MOVJ C00596 BC00596 VJ=30.00
MOVJ C00597 BC00597 VJ=40.00
'**********************
'W18A
'**********************
SFTON P0306
MOVL C00598 BC00598 V=333.3
MOVL C00599 BC00599 V=166.7 PL=0
SFTOF
ARCON
SFTON P0307
MOVL C00600 BC00600 V=10.8
ARCOF
SFTOF
MOVL C00601 BC00601 V=250.0
MOVJ C00602 BC00602 VJ=30.00
MOVJ C00603 BC00603 VJ=30.00
MOVJ C00604 BC00604 VJ=50.00
MOVJ C00605 BC00605 VJ=50.00
MOVJ C00606 BC00606 VJ=50.00
'**********************
'W18B
'**********************
SFTON P0355
MOVL C00607 BC00607 V=166.7
MOVL C00608 BC00608 V=166.7 PL=0
SFTOF
ARCON
SFTON P0354
MOVL C00609 BC00609 V=10.8
ARCOF
MOVL C00610 BC00610 V=250.0
SFTOF
MOVJ C00611 BC00611 VJ=30.00
MOVJ C00612 BC00612 VJ=30.00
MOVJ C00613 BC00613 VJ=40.00
MOVJ C00614 BC00614 VJ=50.00
MOVJ C00615 BC00615 VJ=30.00
'**********************
'W19A
'**********************
MOVL C00616 BC00616 V=166.7
SFTON P0303
MOVL C00617 BC00617 V=166.7 PL=0
SFTOF
ARCON
SFTON P0302
MOVL C00618 BC00618 V=10.8
ARCOF
SFTOF
MOVL C00619 BC00619 V=150.0
MOVJ C00620 BC00620 VJ=30.00
MOVJ C00621 BC00621 VJ=50.00
MOVJ C00622 BC00622 VJ=50.00
'**********************
'W19B
'**********************
SFTON P0358
MOVL C00623 BC00623 V=500.0
MOVL C00624 BC00624 V=166.7 PL=0
SFTOF
ARCON
SFTON P0359
MOVL C00625 BC00625 V=10.8
ARCOF
SFTOF
MOVL C00626 BC00626 V=250.0
MOVJ C00627 BC00627 VJ=40.00
MOVJ C00628 BC00628 VJ=50.00
CALL JOB:MOVE_OUT_OF_TUNNEL
END
